LIN {X 60.580,Y -45.308,Z -141.426,A -90.000,B 90.000,C 0.000} C_DIS
LIN {X 60.651,Y -45.308,Z -141.391,A -90.000,B 90.000,C 0.000} C_DIS
LIN {X 60.882,Y -45.308,Z -141.285,A -90.000,B 90.000,C 0.000} C_DIS
LIN {X 61.927,Y -45.308,Z -140.871,A -90.000,B 90.000,C 0.000} C_DIS
LIN {X 63.864,Y -45.308,Z -140.277,A -90.000,B 90.000,C 0.000} C_DIS
LIN {X 64.038,Y -45.308,Z -140.235,A -90.000,B 90.000,C 0.000} C_DIS
LIN {X 65.559,Y -45.308,Z -140.294,A -90.000,B 90.000,C 0.000} C_DIS
LIN {X 65.640,Y -45.308,Z -140.321,A -90.000,B 90.000,C 0.000} C_DIS
LIN {X 66.939,Y -45.308,Z -140.767,A -90.000,B 90.000,C 0.000} C_DIS
LIN {X 67.087,Y -45.308,Z -140.867,A -90.000,B 90.000,C 0.000} C_DIS
LIN {X 67.673,Y -45.308,Z -141.467,A -90.000,B 90.000,C 0.000} C_DIS
LIN {X 67.788,Y -45.308,Z -141.605,A -90.000,B 90.000,C 0.000} C_DIS
LIN {X 68.275,Y -45.308,Z -142.438,A -90.000,B 90.000,C 0.000} C_DIS
LIN {X 68.917,Y -45.308,Z -143.399,A -90.000,B 90.000,C 0.000} C_DIS
LIN {X 68.990,Y -45.308,Z -143.563,A -90.000,B 90.000,C 0.000} C_DIS
LIN {X 69.573,Y -45.308,Z -144.914,A -90.000,B 90.000,C 0.000} C_DIS
LIN {X 69.855,Y -45.308,Z -145.939,A -90.000,B 90.000,C 0.000} C_DIS
LIN {X 69.892,Y -45.308,Z -146.103,A -90.000,B 90.000,C 0.000} C_DIS
LIN {X 69.904,Y -45.308,Z -146.218,A -90.000,B 90.000,C 0.000} C_DIS
LIN {X 70.372,Y -45.308,Z -149.844,A -90.000,B 90.000,C 0.000} C_DIS
LIN {X 70.397,Y -45.308,Z -150.079,A -90.000,B 90.000,C 0.000} C_DIS
LIN {X 70.477,Y -45.308,Z -152.363,A -90.000,B 90.000,C 0.000} C_DIS
LIN {X 70.544,Y -45.308,Z -153.906,A -90.000,B 90.000,C 0.000} C_DIS
LIN {X 70.353,Y -45.308,Z -157.725,A -90.000,B 90.000,C 0.000} C_DIS
LIN {X 70.338,Y -45.308,Z -157.908,A -90.000,B 90.000,C 0.000} C_DIS
LIN {X 70.199,Y -45.308,Z -158.814,A -90.000,B 90.000,C 0.000} C_DIS
LIN {X 69.684,Y -45.308,Z -161.585,A -90.000,B 90.000,C 0.000} C_DIS
LIN {X 69.620,Y -45.308,Z -161.813,A -90.000,B 90.000,C 0.000} C_DIS
LIN {X 69.546,Y -45.308,Z -162.065,A -90.000,B 90.000,C 0.000} C_DIS
LIN {X 68.616,Y -45.308,Z -165.294,A -90.000,B 90.000,C 0.000} C_DIS
LIN {X 68.534,Y -45.308,Z -165.522,A -90.000,B 90.000,C 0.000} C_DIS
LIN {X 67.458,Y -45.308,Z -168.597,A -90.000,B 90.000,C 0.000} C_DIS
LIN {X 66.943,Y -45.308,Z -170.008,A -90.000,B 90.000,C 0.000} C_DIS
LIN {X 66.324,Y -45.308,Z -171.617,A -90.000,B 90.000,C 0.000} C_DIS
LIN {X 66.282,Y -45.308,Z -171.733,A -90.000,B 90.000,C 0.000} C_DIS
LIN {X 65.339,Y -45.308,Z -174.575,A -90.000,B 90.000,C 0.000} C_DIS
LIN {X 64.922,Y -45.308,Z -176.632,A -90.000,B 90.000,C 0.000} C_DIS
LIN {X 64.757,Y -45.308,Z -177.363,A -90.000,B 90.000,C 0.000} C_DIS
LIN {X 64.366,Y -45.308,Z -180.088,A -90.000,B 90.000,C 0.000} C_DIS
LIN {X 64.330,Y -45.308,Z -180.550,A -90.000,B 90.000,C 0.000} C_DIS
LIN {X 64.152,Y -45.308,Z -182.594,A -90.000,B 90.000,C 0.000} C_DIS
LIN {X 64.105,Y -45.308,Z -183.519,A -90.000,B 90.000,C 0.000} C_DIS
LIN {X 63.918,Y -45.308,Z -186.609,A -90.000,B 90.000,C 0.000} C_DIS
LIN {X 63.839,Y -45.308,Z -187.772,A -90.000,B 90.000,C 0.000} C_DIS
LIN {X 63.829,Y -45.308,Z -187.892,A -90.000,B 90.000,C 0.000} C_DIS
LIN {X 63.562,Y -45.308,Z -190.517,A -90.000,B 90.000,C 0.000} C_DIS
LIN {X 63.102,Y -45.308,Z -193.390,A -90.000,B 90.000,C 0.000} C_DIS
LIN {X 62.752,Y -45.308,Z -194.947,A -90.000,B 90.000,C 0.000} C_DIS
LIN {X 62.328,Y -45.308,Z -196.733,A -90.000,B 90.000,C 0.000} C_DIS
LIN {X 62.297,Y -45.308,Z -196.846,A -90.000,B 90.000,C 0.000} C_DIS
LIN {X 61.644,Y -45.308,Z -199.064,A -90.000,B 90.000,C 0.000} C_DIS
LIN {X 61.144,Y -45.308,Z -200.631,A -90.000,B 90.000,C 0.000} C_DIS
LIN {X 59.629,Y -45.308,Z -204.936,A -90.000,B 90.000,C 0.000} C_DIS
LIN {X 59.533,Y -45.308,Z -205.201,A -90.000,B 90.000,C 0.000} C_DIS
LIN {X 57.775,Y -45.308,Z -209.890,A -90.000,B 90.000,C 0.000} C_DIS
LIN {X 55.827,Y -45.308,Z -214.869,A -90.000,B 90.000,C 0.000} C_DIS
LIN {X 54.437,Y -45.308,Z -218.314,A -90.000,B 90.000,C 0.000} C_DIS
LIN {X 53.740,Y -45.308,Z -220.037,A -90.000,B 90.000,C 0.000} C_DIS
LIN {X 52.345,Y -45.308,Z -223.157,A -90.000,B 90.000,C 0.000} C_DIS
LIN {X 51.395,Y -45.308,Z -225.293,A -90.000,B 90.000,C 0.000} C_DIS
LIN {X 49.882,Y -45.308,Z -228.183,A -90.000,B 90.000,C 0.000} C_DIS
LIN {X 48.676,Y -45.308,Z -230.534,A -90.000,B 90.000,C 0.000} C_DIS
LIN {X 48.535,Y -45.308,Z -230.778,A -90.000,B 90.000,C 0.000} C_DIS
LIN {X 46.664,Y -45.308,Z -233.707,A -90.000,B 90.000,C 0.000} C_DIS
LIN {X 45.317,Y -45.308,Z -235.896,A -90.000,B 90.000,C 0.000} C_DIS
LIN {X 42.480,Y -45.308,Z -239.403,A -90.000,B 90.000,C 0.000} C_DIS
LIN {X 41.445,Y -45.308,Z -240.753,A -90.000,B 90.000,C 0.000} C_DIS
LIN {X 41.263,Y -45.308,Z -240.969,A -90.000,B 90.000,C 0.000} C_DIS
LIN {X 38.792,Y -45.308,Z -243.561,A -90.000,B 90.000,C 0.000} C_DIS
LIN {X 38.792,Y -60.000,Z -243.561,A -90.000,B 90.000,C 0.000} C_DIS
LIN {X -67.298,Y -60.000,Z -243.561,A -90.000,B 90.000,C 0.000} C_DIS
LIN {X -67.298,Y -44.787,Z -243.561,A -90.000,B 90.000,C 0.000} C_DIS
LIN {X -67.270,Y -44.711,Z -243.409,A -90.000,B 90.000,C 0.000} C_DIS
LIN {X -67.144,Y -44.547,Z -243.047,A -90.000,B 90.000,C 0.000} C_DIS
LIN {X -67.046,Y -44.476,Z -242.863,A -90.000,B 90.000,C 0.000} C_DIS
LIN {X -66.669,Y -44.334,Z -242.397,A -90.000,B 90.000,C 0.000} C_DIS
LIN {X -66.161,Y -44.287,Z -242.036,A -90.000,B 90.000,C 0.000} C_DIS
LIN {X -65.652,Y -44.291,Z -241.768,A -90.000,B 90.000,C 0.000} C_DIS
LIN {X -64.439,Y -44.288,Z -241.140,A -90.000,B 90.000,C 0.000} C_DIS
LIN {X -60.910,Y -44.327,Z -239.407,A -90.000,B 90.000,C 0.000} C_DIS
LIN {X -57.171,Y -44.331,Z -237.595,A -90.000,B 90.000,C 0.000} C_DIS
LIN {X -55.898,Y -44.321,Z -236.982,A -90.000,B 90.000,C 0.000} C_DIS
LIN {X -55.409,Y -44.321,Z -236.755,A -90.000,B 90.000,C 0.000} C_DIS
LIN {X -54.668,Y -44.326,Z -236.421,A -90.000,B 90.000,C 0.000} C_DIS
LIN {X -52.760,Y -44.345,Z -235.573,A -90.000,B 90.000,C 0.000} C_DIS
LIN {X -49.209,Y -44.397,Z -234.093,A -90.000,B 90.000,C 0.000} C_DIS
LIN {X -47.684,Y -44.433,Z -233.484,A -90.000,B 90.000,C 0.000} C_DIS
LIN {X -45.954,Y -44.457,Z -232.802,A -90.000,B 90.000,C 0.000} C_DIS
LIN {X -45.316,Y -44.465,Z -232.551,A -90.000,B 90.000,C 0.000} C_DIS
LIN {X -44.202,Y -44.466,Z -232.120,A -90.000,B 90.000,C 0.000} C_DIS
LIN {X -41.863,Y -44.487,Z -231.267,A -90.000,B 90.000,C 0.000} C_DIS
LIN {X -41.293,Y -44.487,Z -231.062,A -90.000,B 90.000,C 0.000} C_DIS
LIN {X -39.930,Y -44.501,Z -230.603,A -90.000,B 90.000,C 0.000} C_DIS
LIN {X -39.608,Y -44.508,Z -230.503,A -90.000,B 90.000,C 0.000} C_DIS
LIN {X -38.618,Y -44.539,Z -230.217,A -90.000,B 90.000,C 0.000} C_DIS
LIN {X -37.408,Y -44.595,Z -229.897,A -90.000,B 90.000,C 0.000} C_DIS
LIN {X -36.049,Y -44.639,Z -229.528,A -90.000,B 90.000,C 0.000} C_DIS
LIN {X -34.932,Y -44.668,Z -229.228,A -90.000,B 90.000,C 0.000} C_DIS
LIN {X -34.798,Y -44.669,Z -229.193,A -90.000,B 90.000,C 0.000} C_DIS
LIN {X -34.317,Y -44.671,Z -229.068,A -90.000,B 90.000,C 0.000} C_DIS
LIN {X -32.516,Y -44.686,Z -228.647,A -90.000,B 90.000,C 0.000} C_DIS
LIN {X -32.064,Y -44.687,Z -228.542,A -90.000,B 90.000,C 0.000} C_DIS
LIN {X -31.983,Y -44.687,Z -228.525,A -90.000,B 90.000,C 0.000} C_DIS
LIN {X -30.904,Y -44.701,Z -228.321,A -90.000,B 90.000,C 0.000} C_DIS
LIN {X -30.738,Y -44.706,Z -228.296,A -90.000,B 90.000,C 0.000} C_DIS
LIN {X -29.560,Y -44.754,Z -228.178,A -90.000,B 90.000,C 0.000} C_DIS
LIN {X -29.093,Y -44.779,Z -228.147,A -90.000,B 90.000,C 0.000} C_DIS
LIN {X -28.473,Y -44.815,Z -228.106,A -90.000,B 90.000,C 0.000} C_DIS
LIN {X -27.647,Y -44.853,Z -228.056,A -90.000,B 90.000,C 0.000} C_DIS
LIN {X -27.097,Y -44.859,Z -228.027,A -90.000,B 90.000,C 0.000} C_DIS
LIN {X -26.119,Y -44.859,Z -227.944,A -90.000,B 90.000,C 0.000} C_DIS
LIN {X -25.569,Y -44.862,Z -227.908,A -90.000,B 90.000,C 0.000} C_DIS
LIN {X -25.234,Y -44.867,Z -227.901,A -90.000,B 90.000,C 0.000} C_DIS
LIN {X -25.053,Y -44.872,Z -227.906,A -90.000,B 90.000,C 0.000} C_DIS
LIN {X -24.470,Y -44.891,Z -227.950,A -90.000,B 90.000,C 0.000} C_DIS
LIN {X -24.240,Y -44.901,Z -227.981,A -90.000,B 90.000,C 0.000} C_DIS
LIN {X -23.242,Y -44.958,Z -228.173,A -90.000,B 90.000,C 0.000} C_DIS
LIN {X -23.055,Y -44.967,Z -228.209,A -90.000,B 90.000,C 0.000} C_DIS
LIN {X -22.552,Y -44.978,Z -228.310,A -90.000,B 90.000,C 0.000} C_DIS
LIN {X -22.026,Y -44.978,Z -228.417,A -90.000,B 90.000,C 0.000} C_DIS
LIN {X -21.725,Y -44.979,Z -228.487,A -90.000,B 90.000,C 0.000} C_DIS
LIN {X -20.617,Y -44.981,Z -228.753,A -90.000,B 90.000,C 0.000} C_DIS
LIN {X -20.425,Y -44.983,Z -228.813,A -90.000,B 90.000,C 0.000} C_DIS
LIN {X -20.250,Y -44.986,Z -228.873,A -90.000,B 90.000,C 0.000} C_DIS
LIN {X -20.100,Y -44.991,Z -228.938,A -90.000,B 90.000,C 0.000} C_DIS
LIN {X -20.052,Y -44.993,Z -228.962,A -90.000,B 90.000,C 0.000} C_DIS
LIN {X -19.857,Y -45.004,Z -229.077,A -90.000,B 90.000,C 0.000} C_DIS
LIN {X -19.708,Y -45.014,Z -229.176,A -90.000,B 90.000,C 0.000} C_DIS
LIN {X -19.467,Y -45.032,Z -229.343,A -90.000,B 90.000,C 0.000} C_DIS
LIN {X -19.339,Y -45.039,Z -229.432,A -90.000,B 90.000,C 0.000} C_DIS
LIN {X -18.431,Y -45.038,Z -230.074,A -90.000,B 90.000,C 0.000} C_DIS
LIN {X -17.329,Y -45.038,Z -230.904,A -90.000,B 90.000,C 0.000} C_DIS
LIN {X -17.131,Y -45.040,Z -231.074,A -90.000,B 90.000,C 0.000} C_DIS
LIN {X -16.995,Y -45.045,Z -231.222,A -90.000,B 90.000,C 0.000} C_DIS
LIN {X -16.869,Y -45.046,Z -231.372,A -90.000,B 90.000,C 0.000} C_DIS
LIN {X -16.752,Y -45.044,Z -231.533,A -90.000,B 90.000,C 0.000} C_DIS
LIN {X -15.804,Y -45.041,Z -233.094,A -90.000,B 90.000,C 0.000} C_DIS
LIN {X -15.426,Y -45.041,Z -233.734,A -90.000,B 90.000,C 0.000} C_DIS
LIN {X -15.257,Y -45.036,Z -234.022,A -90.000,B 90.000,C 0.000} C_DIS
LIN {X -15.172,Y -45.035,Z -234.182,A -90.000,B 90.000,C 0.000} C_DIS
LIN {X -14.961,Y -45.035,Z -234.654,A -90.000,B 90.000,C 0.000} C_DIS
LIN {X -14.274,Y -45.040,Z -236.188,A -90.000,B 90.000,C 0.000} C_DIS
LIN {X -14.110,Y -45.044,Z -236.552,A -90.000,B 90.000,C 0.000} C_DIS
LIN {X -13.993,Y -45.047,Z -236.794,A -90.000,B 90.000,C 0.000} C_DIS
LIN {X -13.255,Y -45.047,Z -238.011,A -90.000,B 90.000,C 0.000} C_DIS
LIN {X -13.065,Y -45.046,Z -238.296,A -90.000,B 90.000,C 0.000} C_DIS
LIN {X -12.733,Y -45.051,Z -238.794,A -90.000,B 90.000,C 0.000} C_DIS
LIN {X -12.646,Y -45.057,Z -238.923,A -90.000,B 90.000,C 0.000} C_DIS
LIN {X -11.097,Y -45.055,Z -240.071,A -90.000,B 90.000,C 0.000} C_DIS
LIN {X -10.769,Y -45.037,Z -240.129,A -90.000,B 90.000,C 0.000} C_DIS
LIN {X -10.257,Y -45.024,Z -240.217,A -90.000,B 90.000,C 0.000} C_DIS
LIN {X -9.508,Y -45.062,Z -240.340,A -90.000,B 90.000,C 0.000} C_DIS
LIN {X -8.784,Y -45.078,Z -240.341,A -90.000,B 90.000,C 0.000} C_DIS
LIN {X -8.272,Y -45.078,Z -240.344,A -90.000,B 90.000,C 0.000} C_DIS
LIN {X -4.569,Y -44.924,Z -239.042,A -90.000,B 90.000,C 0.000} C_DIS
LIN {X -3.870,Y -44.924,Z -238.791,A -90.000,B 90.000,C 0.000} C_DIS
LIN {X -2.390,Y -44.970,Z -238.252,A -90.000,B 90.000,C 0.000} C_DIS
LIN {X -0.853,Y -44.908,Z -236.956,A -90.000,B 90.000,C 0.000} C_DIS
LIN {X -0.001,Y -44.910,Z -236.229,A -90.000,B 90.000,C 0.000} C_DIS
LIN {X 1.219,Y -44.920,Z -235.229,A -90.000,B 90.000,C 0.000} C_DIS
LIN {X 2.676,Y -44.867,Z -233.519,A -90.000,B 90.000,C 0.000} C_DIS
LIN {X 4.369,Y -44.865,Z -231.510,A -90.000,B 90.000,C 0.000} C_DIS
LIN {X 4.575,Y -44.856,Z -231.211,A -90.000,B 90.000,C 0.000} C_DIS
LIN {X 4.834,Y -44.847,Z -230.835,A -90.000,B 90.000,C 0.000} C_DIS
LIN {X 6.303,Y -44.802,Z -228.671,A -90.000,B 90.000,C 0.000} C_DIS
LIN {X 7.363,Y -44.796,Z -227.098,A -90.000,B 90.000,C 0.000} C_DIS
LIN {X 7.515,Y -44.796,Z -226.878,A -90.000,B 90.000,C 0.000} C_DIS
LIN {X 7.864,Y -44.798,Z -226.373,A -90.000,B 90.000,C 0.000} C_DIS
LIN {X 7.939,Y -44.798,Z -226.259,A -90.000,B 90.000,C 0.000} C_DIS
LIN {X 9.938,Y -44.768,Z -222.971,A -90.000,B 90.000,C 0.000} C_DIS
LIN {X 10.445,Y -44.768,Z -222.134,A -90.000,B 90.000,C 0.000} C_DIS
LIN {X 10.596,Y -44.770,Z -221.883,A -90.000,B 90.000,C 0.000} C_DIS
LIN {X 11.790,Y -44.762,Z -219.763,A -90.000,B 90.000,C 0.000} C_DIS
LIN {X 12.145,Y -44.764,Z -219.132,A -90.000,B 90.000,C 0.000} C_DIS
LIN {X 12.682,Y -44.770,Z -218.203,A -90.000,B 90.000,C 0.000} C_DIS
LIN {X 13.008,Y -44.771,Z -217.642,A -90.000,B 90.000,C 0.000} C_DIS
LIN {X 13.171,Y -44.776,Z -217.358,A -90.000,B 90.000,C 0.000} C_DIS
LIN {X 14.056,Y -44.792,Z -215.663,A -90.000,B 90.000,C 0.000} C_DIS
LIN {X 14.543,Y -44.796,Z -214.696,A -90.000,B 90.000,C 0.000} C_DIS
LIN {X 15.364,Y -44.800,Z -213.069,A -90.000,B 90.000,C 0.000} C_DIS
LIN {X 15.477,Y -44.804,Z -212.843,A -90.000,B 90.000,C 0.000} C_DIS
LIN {X 15.756,Y -44.812,Z -212.254,A -90.000,B 90.000,C 0.000} C_DIS
LIN {X 16.265,Y -44.814,Z -211.045,A -90.000,B 90.000,C 0.000} C_DIS
LIN {X 17.100,Y -44.822,Z -209.043,A -90.000,B 90.000,C 0.000} C_DIS
LIN {X 17.373,Y -44.824,Z -208.357,A -90.000,B 90.000,C 0.000} C_DIS
LIN {X 18.130,Y -44.858,Z -206.146,A -90.000,B 90.000,C 0.000} C_DIS
LIN {X 18.726,Y -44.870,Z -204.142,A -90.000,B 90.000,C 0.000} C_DIS
LIN {X 18.849,Y -44.875,Z -203.668,A -90.000,B 90.000,C 0.000} C_DIS
LIN {X 18.987,Y -44.872,Z -202.926,A -90.000,B 90.000,C 0.000} C_DIS
LIN {X 19.274,Y -44.870,Z -201.502,A -90.000,B 90.000,C 0.000} C_DIS
LIN {X 19.608,Y -44.855,Z -199.853,A -90.000,B 90.000,C 0.000} C_DIS
LIN {X 19.652,Y -44.853,Z -199.630,A -90.000,B 90.000,C 0.000} C_DIS
LIN {X 20.199,Y -44.801,Z -196.858,A -90.000,B 90.000,C 0.000} C_DIS
LIN {X 20.446,Y -44.795,Z -195.895,A -90.000,B 90.000,C 0.000} C_DIS
LIN {X 20.541,Y -44.786,Z -195.535,A -90.000,B 90.000,C 0.000} C_DIS
LIN {X 20.564,Y -44.785,Z -195.453,A -90.000,B 90.000,C 0.000} C_DIS
LIN {X 20.642,Y -44.782,Z -195.202,A -90.000,B 90.000,C 0.000} C_DIS
LIN {X 20.915,Y -44.776,Z -194.417,A -90.000,B 90.000,C 0.000} C_DIS
LIN {X 21.045,Y -44.769,Z -194.046,A -90.000,B 90.000,C 0.000} C_DIS
LIN {X 21.881,Y -44.697,Z -191.473,A -90.000,B 90.000,C 0.000} C_DIS
LIN {X 21.929,Y -44.695,Z -191.339,A -90.000,B 90.000,C 0.000} C_DIS
LIN {X 22.045,Y -44.695,Z -191.060,A -90.000,B 90.000,C 0.000} C_DIS
LIN {X 22.081,Y -44.692,Z -190.980,A -90.000,B 90.000,C 0.000} C_DIS
LIN {X 23.068,Y -44.639,Z -188.911,A -90.000,B 90.000,C 0.000} C_DIS
LIN {X 23.201,Y -44.628,Z -188.607,A -90.000,B 90.000,C 0.000} C_DIS
LIN {X 23.652,Y -44.602,Z -187.566,A -90.000,B 90.000,C 0.000} C_DIS
LIN {X 23.710,Y -44.598,Z -187.454,A -90.000,B 90.000,C 0.000} C_DIS
LIN {X 23.765,Y -44.596,Z -187.361,A -90.000,B 90.000,C 0.000} C_DIS
LIN {X 24.257,Y -44.583,Z -186.557,A -90.000,B 90.000,C 0.000} C_DIS
LIN {X 24.363,Y -44.580,Z -186.390,A -90.000,B 90.000,C 0.000} C_DIS
LIN {X 24.685,Y -44.577,Z -185.899,A -90.000,B 90.000,C 0.000} C_DIS
LIN {X 25.700,Y -44.551,Z -184.374,A -90.000,B 90.000,C 0.000} C_DIS
LIN {X 25.827,Y -44.545,Z -184.186,A -90.000,B 90.000,C 0.000} C_DIS
LIN {X 25.890,Y -44.543,Z -184.098,A -90.000,B 90.000,C 0.000} C_DIS
LIN {X 26.870,Y -44.535,Z -182.791,A -90.000,B 90.000,C 0.000} C_DIS
LIN {X 27.875,Y -44.525,Z -181.522,A -90.000,B 90.000,C 0.000} C_DIS
LIN {X 29.146,Y -44.523,Z -179.964,A -90.000,B 90.000,C 0.000} C_DIS
LIN {X 29.462,Y -44.519,Z -179.579,A -90.000,B 90.000,C 0.000} C_DIS
LIN {X 29.729,Y -44.519,Z -179.251,A -90.000,B 90.000,C 0.000} C_DIS
LIN {X 31.269,Y -44.533,Z -177.449,A -90.000,B 90.000,C 0.000} C_DIS
LIN {X 31.603,Y -44.552,Z -177.048,A -90.000,B 90.000,C 0.000} C_DIS
LIN {X 32.293,Y -44.548,Z -176.059,A -90.000,B 90.000,C 0.000} C_DIS
LIN {X 32.817,Y -44.549,Z -175.350,A -90.000,B 90.000,C 0.000} C_DIS
LIN {X 33.023,Y -44.559,Z -175.065,A -90.000,B 90.000,C 0.000} C_DIS
LIN {X 33.889,Y -44.552,Z -173.666,A -90.000,B 90.000,C 0.000} C_DIS
LIN {X 34.095,Y -44.551,Z -173.349,A -90.000,B 90.000,C 0.000} C_DIS
LIN {X 34.249,Y -44.557,Z -173.110,A -90.000,B 90.000,C 0.000} C_DIS
LIN {X 35.410,Y -44.546,Z -171.078,A -90.000,B 90.000,C 0.000} C_DIS
LIN {X 35.530,Y -44.547,Z -170.877,A -90.000,B 90.000,C 0.000} C_DIS
LIN {X 36.271,Y -44.534,Z -169.531,A -90.000,B 90.000,C 0.000} C_DIS
LIN {X 36.563,Y -44.534,Z -169.025,A -90.000,B 90.000,C 0.000} C_DIS
LIN {X 36.810,Y -44.537,Z -168.598,A -90.000,B 90.000,C 0.000} C_DIS
LIN {X 37.039,Y -44.535,Z -168.171,A -90.000,B 90.000,C 0.000} C_DIS
LIN {X 38.276,Y -44.538,Z -166.002,A -90.000,B 90.000,C 0.000} C_DIS
LIN {X 38.520,Y -44.543,Z -165.572,A -90.000,B 90.000,C 0.000} C_DIS
LIN {X 39.176,Y -44.542,Z -164.346,A -90.000,B 90.000,C 0.000} C_DIS
LIN {X 39.927,Y -44.546,Z -163.021,A -90.000,B 90.000,C 0.000} C_DIS
LIN {X 40.188,Y -44.551,Z -162.557,A -90.000,B 90.000,C 0.000} C_DIS
LIN {X 41.605,Y -44.556,Z -159.932,A -90.000,B 90.000,C 0.000} C_DIS
LIN {X 41.932,Y -44.555,Z -159.355,A -90.000,B 90.000,C 0.000} C_DIS
LIN {X 42.596,Y -44.549,Z -158.159,A -90.000,B 90.000,C 0.000} C_DIS
LIN {X 43.799,Y -44.562,Z -156.119,A -90.000,B 90.000,C 0.000} C_DIS
LIN {X 44.380,Y -44.572,Z -155.158,A -90.000,B 90.000,C 0.000} C_DIS
LIN {X 45.309,Y -44.590,Z -153.649,A -90.000,B 90.000,C 0.000} C_DIS
LIN {X 45.559,Y -44.590,Z -153.247,A -90.000,B 90.000,C 0.000} C_DIS
LIN {X 45.740,Y -44.590,Z -152.957,A -90.000,B 90.000,C 0.000} C_DIS
LIN {X 45.907,Y -44.592,Z -152.695,A -90.000,B 90.000,C 0.000} C_DIS
LIN {X 46.546,Y -44.608,Z -151.741,A -90.000,B 90.000,C 0.000} C_DIS
LIN {X 47.431,Y -44.625,Z -150.425,A -90.000,B 90.000,C 0.000} C_DIS
LIN {X 47.669,Y -44.620,Z -150.076,A -90.000,B 90.000,C 0.000} C_DIS
LIN {X 47.901,Y -44.615,Z -149.738,A -90.000,B 90.000,C 0.000} C_DIS
LIN {X 48.068,Y -44.610,Z -149.499,A -90.000,B 90.000,C 0.000} C_DIS
LIN {X 48.191,Y -44.611,Z -149.343,A -90.000,B 90.000,C 0.000} C_DIS
LIN {X 49.907,Y -44.673,Z -147.377,A -90.000,B 90.000,C 0.000} C_DIS
LIN {X 50.941,Y -44.677,Z -146.211,A -90.000,B 90.000,C 0.000} C_DIS
LIN {X 51.066,Y -44.678,Z -146.074,A -90.000,B 90.000,C 0.000} C_DIS
LIN {X 51.221,Y -44.681,Z -145.909,A -90.000,B 90.000,C 0.000} C_DIS
LIN {X 51.436,Y -44.689,Z -145.695,A -90.000,B 90.000,C 0.000} C_DIS
LIN {X 51.619,Y -44.693,Z -145.513,A -90.000,B 90.000,C 0.000} C_DIS
LIN {X 52.346,Y -44.693,Z -144.801,A -90.000,B 90.000,C 0.000} C_DIS
LIN {X 52.988,Y -44.702,Z -144.207,A -90.000,B 90.000,C 0.000} C_DIS
LIN {X 53.091,Y -44.705,Z -144.118,A -90.000,B 90.000,C 0.000} C_DIS
LIN {X 53.267,Y -44.712,Z -143.975,A -90.000,B 90.000,C 0.000} C_DIS
LIN {X 54.172,Y -44.723,Z -143.252,A -90.000,B 90.000,C 0.000} C_DIS
LIN {X 54.518,Y -44.731,Z -142.974,A -90.000,B 90.000,C 0.000} C_DIS
LIN {X 54.749,Y -44.738,Z -142.797,A -90.000,B 90.000,C 0.000} C_DIS
LIN {X 54.837,Y -44.742,Z -142.733,A -90.000,B 90.000,C 0.000} C_DIS
LIN {X 55.082,Y -44.748,Z -142.568,A -90.000,B 90.000,C 0.000} C_DIS
LIN {X 55.785,Y -44.751,Z -142.100,A -90.000,B 90.000,C 0.000} C_DIS
LIN {X 56.241,Y -44.739,Z -141.749,A -90.000,B 90.000,C 0.000} C_DIS
LIN {X 56.322,Y -44.739,Z -141.685,A -90.000,B 90.000,C 0.000} C_DIS
LIN {X 56.542,Y -44.741,Z -141.520,A -90.000,B 90.000,C 0.000} C_DIS
LIN {X 56.749,Y -44.746,Z -141.382,A -90.000,B 90.000,C 0.000} C_DIS
LIN {X 57.457,Y -44.779,Z -140.972,A -90.000,B 90.000,C 0.000} C_DIS
LIN {X 58.083,Y -44.806,Z -140.612,A -90.000,B 90.000,C 0.000} C_DIS
LIN {X 58.544,Y -44.821,Z -140.347,A -90.000,B 90.000,C 0.000} C_DIS
LIN {X 59.599,Y -44.842,Z -139.747,A -90.000,B 90.000,C 0.000} C_DIS
LIN {X 59.775,Y -44.847,Z -139.653,A -90.000,B 90.000,C 0.000} C_DIS
LIN {X 60.047,Y -44.858,Z -139.523,A -90.000,B 90.000,C 0.000} C_DIS
LIN {X 60.145,Y -44.863,Z -139.480,A -90.000,B 90.000,C 0.000} C_DIS
LIN {X 61.205,Y -44.906,Z -139.050,A -90.000,B 90.000,C 0.000} C_DIS
LIN {X 61.325,Y -44.912,Z -139.006,A -90.000,B 90.000,C 0.000} C_DIS
LIN {X 63.019,Y -44.951,Z -138.478,A -90.000,B 90.000,C 0.000} C_DIS
LIN {X 63.286,Y -44.961,Z -138.394,A -90.000,B 90.000,C 0.000} C_DIS
LIN {X 63.399,Y -44.965,Z -138.362,A -90.000,B 90.000,C 0.000} C_DIS
LIN {X 63.573,Y -44.973,Z -138.319,A -90.000,B 90.000,C 0.000} C_DIS
LIN {X 63.859,Y -44.990,Z -138.268,A -90.000,B 90.000,C 0.000} C_DIS
LIN {X 63.954,Y -44.996,Z -138.261,A -90.000,B 90.000,C 0.000} C_DIS
LIN {X 64.116,Y -45.010,Z -138.259,A -90.000,B 90.000,C 0.000} C_DIS
LIN {X 64.331,Y -45.029,Z -138.264,A -90.000,B 90.000,C 0.000} C_DIS
LIN {X 64.863,Y -45.047,Z -138.283,A -90.000,B 90.000,C 0.000} C_DIS
LIN {X 65.684,Y -45.048,Z -138.315,A -90.000,B 90.000,C 0.000} C_DIS
LIN {X 66.179,Y -45.057,Z -138.410,A -90.000,B 90.000,C 0.000} C_DIS
LIN {X 67.117,Y -45.087,Z -138.726,A -90.000,B 90.000,C 0.000} C_DIS
LIN {X 67.287,Y -45.088,Z -138.785,A -90.000,B 90.000,C 0.000} C_DIS
LIN {X 67.593,Y -45.077,Z -138.891,A -90.000,B 90.000,C 0.000} C_DIS
LIN {X 67.764,Y -45.067,Z -138.961,A -90.000,B 90.000,C 0.000} C_DIS
LIN {X 68.013,Y -45.053,Z -139.099,A -90.000,B 90.000,C 0.000} C_DIS
LIN {X 68.201,Y -45.047,Z -139.227,A -90.000,B 90.000,C 0.000} C_DIS
LIN {X 68.448,Y -45.041,Z -139.426,A -90.000,B 90.000,C 0.000} C_DIS
LIN {X 68.506,Y -45.041,Z -139.483,A -90.000,B 90.000,C 0.000} C_DIS
LIN {X 69.091,Y -45.041,Z -140.082,A -90.000,B 90.000,C 0.000} C_DIS
LIN {X 69.156,Y -45.042,Z -140.153,A -90.000,B 90.000,C 0.000} C_DIS
LIN {X 69.272,Y -45.041,Z -140.290,A -90.000,B 90.000,C 0.000} C_DIS
LIN {X 69.341,Y -45.039,Z -140.373,A -90.000,B 90.000,C 0.000} C_DIS
LIN {X 69.430,Y -45.037,Z -140.496,A -90.000,B 90.000,C 0.000} C_DIS
LIN {X 69.500,Y -45.036,Z -140.608,A -90.000,B 90.000,C 0.000} C_DIS
LIN {X 69.955,Y -45.036,Z -141.387,A -90.000,B 90.000,C 0.000} C_DIS
LIN {X 70.098,Y -45.033,Z -141.602,A -90.000,B 90.000,C 0.000} C_DIS
LIN {X 70.558,Y -44.991,Z -142.301,A -90.000,B 90.000,C 0.000} C_DIS
LIN {X 70.720,Y -44.976,Z -142.599,A -90.000,B 90.000,C 0.000} C_DIS
LIN {X 70.739,Y -44.975,Z -142.643,A -90.000,B 90.000,C 0.000} C_DIS
LIN {X 71.371,Y -44.909,Z -144.137,A -90.000,B 90.000,C 0.000} C_DIS
LIN {X 71.460,Y -44.902,Z -144.393,A -90.000,B 90.000,C 0.000} C_DIS
LIN {X 71.742,Y -44.891,Z -145.423,A -90.000,B 90.000,C 0.000} C_DIS
LIN {X 71.765,Y -44.890,Z -145.517,A -90.000,B 90.000,C 0.000} C_DIS
LIN {X 71.801,Y -44.890,Z -145.681,A -90.000,B 90.000,C 0.000} C_DIS
LIN {X 71.836,Y -44.893,Z -145.886,A -90.000,B 90.000,C 0.000} C_DIS
LIN {X 71.845,Y -44.894,Z -145.968,A -90.000,B 90.000,C 0.000} C_DIS
LIN {X 71.894,Y -44.901,Z -146.336,A -90.000,B 90.000,C 0.000} C_DIS
LIN {X 72.312,Y -44.890,Z -149.594,A -90.000,B 90.000,C 0.000} C_DIS
LIN {X 72.342,Y -44.890,Z -149.873,A -90.000,B 90.000,C 0.000} C_DIS
LIN {X 72.352,Y -44.891,Z -150.010,A -90.000,B 90.000,C 0.000} C_DIS
LIN {X 72.365,Y -44.896,Z -150.357,A -90.000,B 90.000,C 0.000} C_DIS
LIN {X 72.425,Y -44.862,Z -152.273,A -90.000,B 90.000,C 0.000} C_DIS
LIN {X 72.484,Y -44.830,Z -153.823,A -90.000,B 90.000,C 0.000} C_DIS
LIN {X 72.483,Y -44.829,Z -154.003,A -90.000,B 90.000,C 0.000} C_DIS
LIN {X 72.473,Y -44.829,Z -154.206,A -90.000,B 90.000,C 0.000} C_DIS
LIN {X 72.280,Y -44.780,Z -157.815,A -90.000,B 90.000,C 0.000} C_DIS
LIN {X 72.259,Y -44.778,Z -158.070,A -90.000,B 90.000,C 0.000} C_DIS
LIN {X 72.244,Y -44.778,Z -158.201,A -90.000,B 90.000,C 0.000} C_DIS
LIN {X 72.103,Y -44.771,Z -159.107,A -90.000,B 90.000,C 0.000} C_DIS
LIN {X 71.586,Y -44.771,Z -161.895,A -90.000,B 90.000,C 0.000} C_DIS
LIN {X 71.567,Y -44.769,Z -161.987,A -90.000,B 90.000,C 0.000} C_DIS
LIN {X 71.533,Y -44.768,Z -162.121,A -90.000,B 90.000,C 0.000} C_DIS
LIN {X 71.395,Y -44.767,Z -162.602,A -90.000,B 90.000,C 0.000} C_DIS
LIN {X 70.529,Y -44.765,Z -165.605,A -90.000,B 90.000,C 0.000} C_DIS
LIN {X 70.465,Y -44.761,Z -165.826,A -90.000,B 90.000,C 0.000} C_DIS
LIN {X 70.427,Y -44.760,Z -165.943,A -90.000,B 90.000,C 0.000} C_DIS
LIN {X 70.347,Y -44.760,Z -166.164,A -90.000,B 90.000,C 0.000} C_DIS
LIN {X 69.884,Y -44.757,Z -167.486,A -90.000,B 90.000,C 0.000} C_DIS
LIN {X 69.386,Y -44.757,Z -168.908,A -90.000,B 90.000,C 0.000} C_DIS
LIN {X 69.272,Y -44.755,Z -169.232,A -90.000,B 90.000,C 0.000} C_DIS
LIN {X 68.748,Y -44.753,Z -170.667,A -90.000,B 90.000,C 0.000} C_DIS
LIN {X 68.220,Y -44.759,Z -172.045,A -90.000,B 90.000,C 0.000} C_DIS
LIN {X 68.100,Y -44.764,Z -172.364,A -90.000,B 90.000,C 0.000} C_DIS
LIN {X 67.259,Y -44.767,Z -174.903,A -90.000,B 90.000,C 0.000} C_DIS
LIN {X 67.204,Y -44.771,Z -175.071,A -90.000,B 90.000,C 0.000} C_DIS
LIN {X 66.811,Y -44.762,Z -176.996,A -90.000,B 90.000,C 0.000} C_DIS
LIN {X 66.651,Y -44.763,Z -177.711,A -90.000,B 90.000,C 0.000} C_DIS
LIN {X 66.420,Y -44.767,Z -179.327,A -90.000,B 90.000,C 0.000} C_DIS
LIN {X 66.281,Y -44.767,Z -180.299,A -90.000,B 90.000,C 0.000} C_DIS
LIN {X 66.272,Y -44.765,Z -180.412,A -90.000,B 90.000,C 0.000} C_DIS
LIN {X 66.077,Y -44.769,Z -182.692,A -90.000,B 90.000,C 0.000} C_DIS
LIN {X 66.063,Y -44.768,Z -182.930,A -90.000,B 90.000,C 0.000} C_DIS
LIN {X 66.029,Y -44.768,Z -183.603,A -90.000,B 90.000,C 0.000} C_DIS
LIN {X 65.918,Y -44.772,Z -185.458,A -90.000,B 90.000,C 0.000} C_DIS
LIN {X 65.848,Y -44.769,Z -186.602,A -90.000,B 90.000,C 0.000} C_DIS
LIN {X 65.772,Y -44.765,Z -187.735,A -90.000,B 90.000,C 0.000} C_DIS
LIN {X 65.745,Y -44.760,Z -188.054,A -90.000,B 90.000,C 0.000} C_DIS
LIN {X 65.460,Y -44.708,Z -190.715,A -90.000,B 90.000,C 0.000} C_DIS
LIN {X 65.446,Y -44.706,Z -190.818,A -90.000,B 90.000,C 0.000} C_DIS
LIN {X 65.426,Y -44.706,Z -190.942,A -90.000,B 90.000,C 0.000} C_DIS
LIN {X 65.314,Y -44.693,Z -191.614,A -90.000,B 90.000,C 0.000} C_DIS
LIN {X 64.970,Y -44.658,Z -193.689,A -90.000,B 90.000,C 0.000} C_DIS
LIN {X 64.947,Y -44.657,Z -193.806,A -90.000,B 90.000,C 0.000} C_DIS
LIN {X 64.588,Y -44.634,Z -195.361,A -90.000,B 90.000,C 0.000} C_DIS
LIN {X 64.158,Y -44.617,Z -197.149,A -90.000,B 90.000,C 0.000} C_DIS
LIN {X 64.118,Y -44.614,Z -197.297,A -90.000,B 90.000,C 0.000} C_DIS
LIN {X 63.435,Y -44.594,Z -199.592,A -90.000,B 90.000,C 0.000} C_DIS
LIN {X 63.229,Y -44.594,Z -200.242,A -90.000,B 90.000,C 0.000} C_DIS
LIN {X 62.984,Y -44.594,Z -201.009,A -90.000,B 90.000,C 0.000} C_DIS
LIN {X 62.923,Y -44.592,Z -201.198,A -90.000,B 90.000,C 0.000} C_DIS
LIN {X 61.464,Y -44.590,Z -205.345,A -90.000,B 90.000,C 0.000} C_DIS
LIN {X 61.299,Y -44.589,Z -205.805,A -90.000,B 90.000,C 0.000} C_DIS
LIN {X 59.522,Y -44.587,Z -210.545,A -90.000,B 90.000,C 0.000} C_DIS
LIN {X 57.563,Y -44.586,Z -215.548,A -90.000,B 90.000,C 0.000} C_DIS
LIN {X 56.526,Y -44.585,Z -218.119,A -90.000,B 90.000,C 0.000} C_DIS
LIN {X 55.553,Y -44.585,Z -220.526,A -90.000,B 90.000,C 0.000} C_DIS
LIN {X 55.467,Y -44.582,Z -220.736,A -90.000,B 90.000,C 0.000} C_DIS
LIN {X 54.511,Y -44.582,Z -222.879,A -90.000,B 90.000,C 0.000} C_DIS
LIN {X 53.209,Y -44.583,Z -225.799,A -90.000,B 90.000,C 0.000} C_DIS
LIN {X 53.095,Y -44.577,Z -226.050,A -90.000,B 90.000,C 0.000} C_DIS
LIN {X 53.057,Y -44.576,Z -226.130,A -90.000,B 90.000,C 0.000} C_DIS
LIN {X 51.538,Y -44.585,Z -229.041,A -90.000,B 90.000,C 0.000} C_DIS
LIN {X 50.499,Y -44.585,Z -231.064,A -90.000,B 90.000,C 0.000} C_DIS
LIN {X 50.431,Y -44.582,Z -231.194,A -90.000,B 90.000,C 0.000} C_DIS
LIN {X 50.303,Y -44.576,Z -231.436,A -90.000,B 90.000,C 0.000} C_DIS
LIN {X 50.122,Y -44.572,Z -231.747,A -90.000,B 90.000,C 0.000} C_DIS
LIN {X 48.254,Y -44.592,Z -234.687,A -90.000,B 90.000,C 0.000} C_DIS
LIN {X 47.161,Y -44.592,Z -236.462,A -90.000,B 90.000,C 0.000} C_DIS
LIN {X 46.922,Y -44.572,Z -236.836,A -90.000,B 90.000,C 0.000} C_DIS
LIN {X 46.845,Y -44.568,Z -236.954,A -90.000,B 90.000,C 0.000} C_DIS
LIN {X 46.776,Y -44.568,Z -237.046,A -90.000,B 90.000,C 0.000} C_DIS
LIN {X 43.977,Y -44.606,Z -240.530,A -90.000,B 90.000,C 0.000} C_DIS
LIN {X 43.325,Y -44.606,Z -241.379,A -90.000,B 90.000,C 0.000} C_DIS
LIN {X 43.161,Y -44.602,Z -241.591,A -90.000,B 90.000,C 0.000} C_DIS
LIN {X 42.926,Y -44.589,Z -241.888,A -90.000,B 90.000,C 0.000} C_DIS
LIN {X 42.871,Y -44.586,Z -241.956,A -90.000,B 90.000,C 0.000} C_DIS
LIN {X 42.687,Y -44.580,Z -242.170,A -90.000,B 90.000,C 0.000} C_DIS
LIN {X 42.611,Y -44.579,Z -242.254,A -90.000,B 90.000,C 0.000} C_DIS
LIN {X 41.925,Y -44.579,Z -242.974,A -90.000,B 90.000,C 0.000} C_DIS
LIN {X 41.369,Y -44.587,Z -243.561,A -90.000,B 90.000,C 0.000} C_DIS
LIN {X 41.369,Y -60.000,Z -243.561,A -90.000,B 90.000,C 0.000} C_DIS
LIN {X -56.008,Y -60.000,Z -235.133,A -90.000,B 90.000,C 0.000} C_DIS
LIN {X -56.008,Y -43.308,Z -235.133,A -90.000,B 90.000,C 0.000} C_DIS
LIN {X -55.361,Y -43.318,Z -234.839,A -90.000,B 90.000,C 0.000} C_DIS
LIN {X -53.415,Y -43.352,Z -233.966,A -90.000,B 90.000,C 0.000} C_DIS
LIN {X -52.543,Y -43.378,Z -233.594,A -90.000,B 90.000,C 0.000} C_DIS
LIN {X -51.053,Y -43.410,Z -232.966,A -90.000,B 90.000,C 0.000} C_DIS
LIN {X -49.827,Y -43.429,Z -232.455,A -90.000,B 90.000,C 0.000} C_DIS
LIN {X -45.890,Y -43.522,Z -230.883,A -90.000,B 90.000,C 0.000} C_DIS
LIN {X -44.802,Y -43.537,Z -230.453,A -90.000,B 90.000,C 0.000} C_DIS
LIN {X -41.858,Y -43.612,Z -229.355,A -90.000,B 90.000,C 0.000} C_DIS
LIN {X -40.787,Y -43.652,Z -228.979,A -90.000,B 90.000,C 0.000} C_DIS
LIN {X -40.453,Y -43.666,Z -228.862,A -90.000,B 90.000,C 0.000} C_DIS
LIN {X -40.090,Y -43.683,Z -228.746,A -90.000,B 90.000,C 0.000} C_DIS
LIN {X -39.516,Y -43.713,Z -228.574,A -90.000,B 90.000,C 0.000} C_DIS
LIN {X -39.050,Y -43.730,Z -228.439,A -90.000,B 90.000,C 0.000} C_DIS
LIN {X -37.852,Y -43.785,Z -228.123,A -90.000,B 90.000,C 0.000} C_DIS
LIN {X -35.704,Y -43.873,Z -227.532,A -90.000,B 90.000,C 0.000} C_DIS
LIN {X -34.731,Y -43.905,Z -227.267,A -90.000,B 90.000,C 0.000} C_DIS
LIN {X -32.446,Y -44.000,Z -226.703,A -90.000,B 90.000,C 0.000} C_DIS
LIN {X -32.324,Y -44.006,Z -226.676,A -90.000,B 90.000,C 0.000} C_DIS
LIN {X -31.694,Y -44.042,Z -226.547,A -90.000,B 90.000,C 0.000} C_DIS
LIN {X -31.250,Y -44.067,Z -226.456,A -90.000,B 90.000,C 0.000} C_DIS
LIN {X -31.001,Y -44.085,Z -226.413,A -90.000,B 90.000,C 0.000} C_DIS
LIN {X -30.903,Y -44.093,Z -226.399,A -90.000,B 90.000,C 0.000} C_DIS
LIN {X -30.749,Y -44.102,Z -226.383,A -90.000,B 90.000,C 0.000} C_DIS
LIN {X -29.657,Y -44.157,Z -226.272,A -90.000,B 90.000,C 0.000} C_DIS
LIN {X -28.562,Y -44.223,Z -226.198,A -90.000,B 90.000,C 0.000} C_DIS
LIN {X -27.339,Y -44.297,Z -226.117,A -90.000,B 90.000,C 0.000} C_DIS
LIN {X -27.223,Y -44.303,Z -226.110,A -90.000,B 90.000,C 0.000} C_DIS
LIN {X -26.196,Y -44.349,Z -226.011,A -90.000,B 90.000,C 0.000} C_DIS
LIN {X -25.626,Y -44.379,Z -225.968,A -90.000,B 90.000,C 0.000} C_DIS
LIN {X -25.219,Y -44.401,Z -225.956,A -90.000,B 90.000,C 0.000} C_DIS
LIN {X -24.916,Y -44.422,Z -225.962,A -90.000,B 90.000,C 0.000} C_DIS
LIN {X -24.803,Y -44.431,Z -225.970,A -90.000,B 90.000,C 0.000} C_DIS
LIN {X -24.278,Y -44.451,Z -226.009,A -90.000,B 90.000,C 0.000} C_DIS
LIN {X -23.941,Y -44.467,Z -226.051,A -90.000,B 90.000,C 0.000} C_DIS
LIN {X -23.762,Y -44.478,Z -226.083,A -90.000,B 90.000,C 0.000} C_DIS
LIN {X -21.576,Y -44.604,Z -226.504,A -90.000,B 90.000,C 0.000} C_DIS
LIN {X -21.265,Y -44.624,Z -226.574,A -90.000,B 90.000,C 0.000} C_DIS
LIN {X -20.982,Y -44.639,Z -226.639,A -90.000,B 90.000,C 0.000} C_DIS
LIN {X -20.471,Y -44.653,Z -226.759,A -90.000,B 90.000,C 0.000} C_DIS
LIN {X -20.157,Y -44.655,Z -226.834,A -90.000,B 90.000,C 0.000} C_DIS
LIN {X -20.020,Y -44.658,Z -226.871,A -90.000,B 90.000,C 0.000} C_DIS
LIN {X -19.768,Y -44.663,Z -226.951,A -90.000,B 90.000,C 0.000} C_DIS
LIN {X -19.594,Y -44.667,Z -227.011,A -90.000,B 90.000,C 0.000} C_DIS
LIN {X -19.497,Y -44.670,Z -227.047,A -90.000,B 90.000,C 0.000} C_DIS
LIN {X -19.281,Y -44.678,Z -227.140,A -90.000,B 90.000,C 0.000} C_DIS
LIN {X -19.160,Y -44.684,Z -227.199,A -90.000,B 90.000,C 0.000} C_DIS
LIN {X -19.089,Y -44.687,Z -227.236,A -90.000,B 90.000,C 0.000} C_DIS
LIN {X -18.836,Y -44.702,Z -227.384,A -90.000,B 90.000,C 0.000} C_DIS
LIN {X -18.671,Y -44.714,Z -227.490,A -90.000,B 90.000,C 0.000} C_DIS
LIN {X -18.447,Y -44.730,Z -227.643,A -90.000,B 90.000,C 0.000} C_DIS
LIN {X -17.850,Y -44.775,Z -228.057,A -90.000,B 90.000,C 0.000} C_DIS
LIN {X -17.721,Y -44.781,Z -228.147,A -90.000,B 90.000,C 0.000} C_DIS
LIN {X -17.238,Y -44.781,Z -228.489,A -90.000,B 90.000,C 0.000} C_DIS
LIN {X -16.136,Y -44.782,Z -229.319,A -90.000,B 90.000,C 0.000} C_DIS
LIN {X -16.033,Y -44.782,Z -229.402,A -90.000,B 90.000,C 0.000} C_DIS
LIN {X -15.835,Y -44.784,Z -229.572,A -90.000,B 90.000,C 0.000} C_DIS
LIN {X -15.690,Y -44.787,Z -229.711,A -90.000,B 90.000,C 0.000} C_DIS
LIN {X -15.533,Y -44.792,Z -229.881,A -90.000,B 90.000,C 0.000} C_DIS
LIN {X -15.451,Y -44.796,Z -229.975,A -90.000,B 90.000,C 0.000} C_DIS
LIN {X -15.336,Y -44.796,Z -230.112,A -90.000,B 90.000,C 0.000} C_DIS
LIN {X -15.269,Y -44.793,Z -230.200,A -90.000,B 90.000,C 0.000} C_DIS
LIN {X -15.152,Y -44.789,Z -230.360,A -90.000,B 90.000,C 0.000} C_DIS
LIN {X -15.056,Y -44.787,Z -230.504,A -90.000,B 90.000,C 0.000} C_DIS
LIN {X -14.501,Y -44.776,Z -231.422,A -90.000,B 90.000,C 0.000} C_DIS
LIN {X -14.098,Y -44.775,Z -232.086,A -90.000,B 90.000,C 0.000} C_DIS
LIN {X -13.890,Y -44.774,Z -232.438,A -90.000,B 90.000,C 0.000} C_DIS
LIN {X -13.598,Y -44.767,Z -232.934,A -90.000,B 90.000,C 0.000} C_DIS
LIN {X -13.547,Y -44.766,Z -233.021,A -90.000,B 90.000,C 0.000} C_DIS
LIN {X -13.414,Y -44.765,Z -233.268,A -90.000,B 90.000,C 0.000} C_DIS
LIN {X -13.364,Y -44.765,Z -233.371,A -90.000,B 90.000,C 0.000} C_DIS
LIN {X -12.618,Y -44.773,Z -235.036,A -90.000,B 90.000,C 0.000} C_DIS
LIN {X -12.312,Y -44.785,Z -235.717,A -90.000,B 90.000,C 0.000} C_DIS
LIN {X -12.247,Y -44.787,Z -235.851,A -90.000,B 90.000,C 0.000} C_DIS
LIN {X -12.160,Y -44.787,Z -235.993,A -90.000,B 90.000,C 0.000} C_DIS
LIN {X -11.579,Y -44.802,Z -236.946,A -90.000,B 90.000,C 0.000} C_DIS
LIN {X -11.233,Y -44.808,Z -237.465,A -90.000,B 90.000,C 0.000} C_DIS
LIN {X -11.186,Y -44.811,Z -237.535,A -90.000,B 90.000,C 0.000} C_DIS
LIN {X -10.296,Y -44.811,Z -238.194,A -90.000,B 90.000,C 0.000} C_DIS
LIN {X -10.132,Y -44.801,Z -238.223,A -90.000,B 90.000,C 0.000} C_DIS
LIN {X -9.335,Y -44.782,Z -238.360,A -90.000,B 90.000,C 0.000} C_DIS
LIN {X -8.611,Y -44.753,Z -238.369,A -90.000,B 90.000,C 0.000} C_DIS
LIN {X -8.113,Y -44.713,Z -238.197,A -90.000,B 90.000,C 0.000} C_DIS
LIN {X -6.122,Y -44.631,Z -237.497,A -90.000,B 90.000,C 0.000} C_DIS
LIN {X -3.794,Y -44.610,Z -236.666,A -90.000,B 90.000,C 0.000} C_DIS
LIN {X -3.394,Y -44.623,Z -236.520,A -90.000,B 90.000,C 0.000} C_DIS
LIN {X -1.244,Y -44.538,Z -234.707,A -90.000,B 90.000,C 0.000} C_DIS
LIN {X -0.656,Y -44.519,Z -234.230,A -90.000,B 90.000,C 0.000} C_DIS
LIN {X -0.339,Y -44.513,Z -233.973,A -90.000,B 90.000,C 0.000} C_DIS
LIN {X -0.161,Y -44.516,Z -233.827,A -90.000,B 90.000,C 0.000} C_DIS
LIN {X 2.815,Y -44.409,Z -230.331,A -90.000,B 90.000,C 0.000} C_DIS
LIN {X 3.065,Y -44.392,Z -229.972,A -90.000,B 90.000,C 0.000} C_DIS
LIN {X 4.406,Y -44.354,Z -227.999,A -90.000,B 90.000,C 0.000} C_DIS
LIN {X 5.766,Y -44.315,Z -225.995,A -90.000,B 90.000,C 0.000} C_DIS
LIN {X 5.942,Y -44.312,Z -225.742,A -90.000,B 90.000,C 0.000} C_DIS
LIN {X 6.278,Y -44.311,Z -225.254,A -90.000,B 90.000,C 0.000} C_DIS
LIN {X 6.791,Y -44.297,Z -224.416,A -90.000,B 90.000,C 0.000} C_DIS
LIN {X 8.668,Y -44.280,Z -221.323,A -90.000,B 90.000,C 0.000} C_DIS
LIN {X 8.923,Y -44.285,Z -220.900,A -90.000,B 90.000,C 0.000} C_DIS
LIN {X 9.741,Y -44.288,Z -219.444,A -90.000,B 90.000,C 0.000} C_DIS
LIN {X 10.467,Y -44.279,Z -218.158,A -90.000,B 90.000,C 0.000} C_DIS
LIN {X 11.210,Y -44.276,Z -216.879,A -90.000,B 90.000,C 0.000} C_DIS
LIN {X 11.473,Y -44.286,Z -216.421,A -90.000,B 90.000,C 0.000} C_DIS
LIN {X 12.353,Y -44.297,Z -214.737,A -90.000,B 90.000,C 0.000} C_DIS
LIN {X 12.438,Y -44.297,Z -214.567,A -90.000,B 90.000,C 0.000} C_DIS
LIN {X 13.521,Y -44.334,Z -212.403,A -90.000,B 90.000,C 0.000} C_DIS
LIN {X 13.729,Y -44.345,Z -211.985,A -90.000,B 90.000,C 0.000} C_DIS
LIN {X 13.979,Y -44.357,Z -211.456,A -90.000,B 90.000,C 0.000} C_DIS
LIN {X 14.466,Y -44.373,Z -210.290,A -90.000,B 90.000,C 0.000} C_DIS
LIN {X 15.289,Y -44.404,Z -208.303,A -90.000,B 90.000,C 0.000} C_DIS
LIN {X 15.461,Y -44.410,Z -207.870,A -90.000,B 90.000,C 0.000} C_DIS
LIN {X 15.539,Y -44.415,Z -207.672,A -90.000,B 90.000,C 0.000} C_DIS
LIN {X 16.267,Y -44.443,Z -205.546,A -90.000,B 90.000,C 0.000} C_DIS
LIN {X 16.843,Y -44.451,Z -203.614,A -90.000,B 90.000,C 0.000} C_DIS
LIN {X 16.940,Y -44.451,Z -203.242,A -90.000,B 90.000,C 0.000} C_DIS
LIN {X 17.073,Y -44.441,Z -202.541,A -90.000,B 90.000,C 0.000} C_DIS
LIN {X 17.564,Y -44.413,Z -200.127,A -90.000,B 90.000,C 0.000} C_DIS
LIN {X 17.720,Y -44.392,Z -199.373,A -90.000,B 90.000,C 0.000} C_DIS
LIN {X 17.850,Y -44.371,Z -198.723,A -90.000,B 90.000,C 0.000} C_DIS
LIN {X 18.306,Y -44.272,Z -196.484,A -90.000,B 90.000,C 0.000} C_DIS
LIN {X 18.331,Y -44.268,Z -196.381,A -90.000,B 90.000,C 0.000} C_DIS
LIN {X 18.693,Y -44.226,Z -195.015,A -90.000,B 90.000,C 0.000} C_DIS
LIN {X 18.732,Y -44.223,Z -194.882,A -90.000,B 90.000,C 0.000} C_DIS
LIN {X 18.830,Y -44.212,Z -194.575,A -90.000,B 90.000,C 0.000} C_DIS
LIN {X 19.230,Y -44.181,Z -193.446,A -90.000,B 90.000,C 0.000} C_DIS
LIN {X 19.272,Y -44.176,Z -193.320,A -90.000,B 90.000,C 0.000} C_DIS
LIN {X 20.103,Y -44.035,Z -190.839,A -90.000,B 90.000,C 0.000} C_DIS
LIN {X 20.155,Y -44.029,Z -190.700,A -90.000,B 90.000,C 0.000} C_DIS
LIN {X 20.189,Y -44.026,Z -190.616,A -90.000,B 90.000,C 0.000} C_DIS
LIN {X 20.340,Y -44.017,Z -190.265,A -90.000,B 90.000,C 0.000} C_DIS
LIN {X 20.376,Y -44.014,Z -190.185,A -90.000,B 90.000,C 0.000} C_DIS
LIN {X 21.365,Y -43.910,Z -188.156,A -90.000,B 90.000,C 0.000} C_DIS
LIN {X 21.667,Y -43.868,Z -187.485,A -90.000,B 90.000,C 0.000} C_DIS
LIN {X 21.912,Y -43.840,Z -186.933,A -90.000,B 90.000,C 0.000} C_DIS
LIN {X 21.961,Y -43.834,Z -186.823,A -90.000,B 90.000,C 0.000} C_DIS
LIN {X 22.069,Y -43.827,Z -186.610,A -90.000,B 90.000,C 0.000} C_DIS
LIN {X 22.173,Y -43.823,Z -186.429,A -90.000,B 90.000,C 0.000} C_DIS
LIN {X 22.775,Y -43.793,Z -185.462,A -90.000,B 90.000,C 0.000} C_DIS
LIN {X 23.162,Y -43.769,Z -184.884,A -90.000,B 90.000,C 0.000} C_DIS
LIN {X 24.098,Y -43.718,Z -183.502,A -90.000,B 90.000,C 0.000} C_DIS
LIN {X 24.342,Y -43.701,Z -183.147,A -90.000,B 90.000,C 0.000} C_DIS
LIN {X 24.448,Y -43.697,Z -183.001,A -90.000,B 90.000,C 0.000} C_DIS
LIN {X 24.690,Y -43.690,Z -182.682,A -90.000,B 90.000,C 0.000} C_DIS
LIN {X 25.459,Y -43.655,Z -181.680,A -90.000,B 90.000,C 0.000} C_DIS
LIN {X 26.489,Y -43.628,Z -180.392,A -90.000,B 90.000,C 0.000} C_DIS
LIN {X 27.452,Y -43.613,Z -179.223,A -90.000,B 90.000,C 0.000} C_DIS
LIN {X 27.965,Y -43.604,Z -178.601,A -90.000,B 90.000,C 0.000} C_DIS
LIN {X 28.381,Y -43.602,Z -178.093,A -90.000,B 90.000,C 0.000} C_DIS
LIN {X 29.602,Y -43.615,Z -176.662,A -90.000,B 90.000,C 0.000} C_DIS
LIN {X 30.192,Y -43.648,Z -175.952,A -90.000,B 90.000,C 0.000} C_DIS
LIN {X 30.532,Y -43.642,Z -175.469,A -90.000,B 90.000,C 0.000} C_DIS
LIN {X 30.863,Y -43.634,Z -175.002,A -90.000,B 90.000,C 0.000} C_DIS
LIN {X 31.081,Y -43.633,Z -174.707,A -90.000,B 90.000,C 0.000} C_DIS
LIN {X 31.546,Y -43.654,Z -174.062,A -90.000,B 90.000,C 0.000} C_DIS
LIN {X 32.224,Y -43.641,Z -172.975,A -90.000,B 90.000,C 0.000} C_DIS
LIN {X 32.409,Y -43.634,Z -172.683,A -90.000,B 90.000,C 0.000} C_DIS
LIN {X 32.464,Y -43.633,Z -172.598,A -90.000,B 90.000,C 0.000} C_DIS
LIN {X 32.732,Y -43.641,Z -172.181,A -90.000,B 90.000,C 0.000} C_DIS
LIN {X 33.770,Y -43.616,Z -170.378,A -90.000,B 90.000,C 0.000} C_DIS
LIN {X 33.894,Y -43.616,Z -170.162,A -90.000,B 90.000,C 0.000} C_DIS
LIN {X 33.993,Y -43.618,Z -169.995,A -90.000,B 90.000,C 0.000} C_DIS
LIN {X 34.740,Y -43.600,Z -168.644,A -90.000,B 90.000,C 0.000} C_DIS
LIN {X 35.045,Y -43.600,Z -168.118,A -90.000,B 90.000,C 0.000} C_DIS
LIN {X 35.265,Y -43.604,Z -167.737,A -90.000,B 90.000,C 0.000} C_DIS
LIN {X 35.504,Y -43.599,Z -167.295,A -90.000,B 90.000,C 0.000} C_DIS
LIN {X 36.493,Y -43.603,Z -165.559,A -90.000,B 90.000,C 0.000} C_DIS
LIN {X 36.970,Y -43.614,Z -164.714,A -90.000,B 90.000,C 0.000} C_DIS
LIN {X 37.384,Y -43.612,Z -163.943,A -90.000,B 90.000,C 0.000} C_DIS
LIN {X 37.638,Y -43.610,Z -163.472,A -90.000,B 90.000,C 0.000} C_DIS
LIN {X 38.115,Y -43.617,Z -162.624,A -90.000,B 90.000,C 0.000} C_DIS
LIN {X 38.634,Y -43.632,Z -161.694,A -90.000,B 90.000,C 0.000} C_DIS
LIN {X 39.983,Y -43.646,Z -159.187,A -90.000,B 90.000,C 0.000} C_DIS
LIN {X 40.055,Y -43.647,Z -159.055,A -90.000,B 90.000,C 0.000} C_DIS
LIN {X 40.374,Y -43.653,Z -158.484,A -90.000,B 90.000,C 0.000} C_DIS
LIN {X 41.055,Y -43.661,Z -157.245,A -90.000,B 90.000,C 0.000} C_DIS
LIN {X 41.378,Y -43.672,Z -156.691,A -90.000,B 90.000,C 0.000} C_DIS
LIN {X 42.260,Y -43.697,Z -155.179,A -90.000,B 90.000,C 0.000} C_DIS
LIN {X 42.920,Y -43.722,Z -154.078,A -90.000,B 90.000,C 0.000} C_DIS
LIN {X 43.378,Y -43.740,Z -153.326,A -90.000,B 90.000,C 0.000} C_DIS
LIN {X 43.921,Y -43.758,Z -152.438,A -90.000,B 90.000,C 0.000} C_DIS
LIN {X 44.208,Y -43.765,Z -151.971,A -90.000,B 90.000,C 0.000} C_DIS
LIN {X 44.398,Y -43.772,Z -151.671,A -90.000,B 90.000,C 0.000} C_DIS
LIN {X 45.149,Y -43.810,Z -150.534,A -90.000,B 90.000,C 0.000} C_DIS
LIN {X 45.392,Y -43.816,Z -150.171,A -90.000,B 90.000,C 0.000} C_DIS
LIN {X 45.916,Y -43.816,Z -149.400,A -90.000,B 90.000,C 0.000} C_DIS
LIN {X 46.553,Y -43.816,Z -148.461,A -90.000,B 90.000,C 0.000} C_DIS
LIN {X 46.634,Y -43.818,Z -148.351,A -90.000,B 90.000,C 0.000} C_DIS
LIN {X 46.756,Y -43.823,Z -148.194,A -90.000,B 90.000,C 0.000} C_DIS
LIN {X 46.818,Y -43.827,Z -148.119,A -90.000,B 90.000,C 0.000} C_DIS
LIN {X 47.618,Y -43.886,Z -147.183,A -90.000,B 90.000,C 0.000} C_DIS
LIN {X 48.834,Y -43.936,Z -145.785,A -90.000,B 90.000,C 0.000} C_DIS
LIN {X 49.603,Y -43.952,Z -144.912,A -90.000,B 90.000,C 0.000} C_DIS
LIN {X 49.868,Y -43.956,Z -144.627,A -90.000,B 90.000,C 0.000} C_DIS
LIN {X 50.405,Y -43.975,Z -144.089,A -90.000,B 90.000,C 0.000} C_DIS
LIN {X 50.709,Y -43.980,Z -143.788,A -90.000,B 90.000,C 0.000} C_DIS
LIN {X 51.082,Y -43.984,Z -143.423,A -90.000,B 90.000,C 0.000} C_DIS
LIN {X 51.773,Y -44.001,Z -142.782,A -90.000,B 90.000,C 0.000} C_DIS
LIN {X 51.928,Y -44.007,Z -142.648,A -90.000,B 90.000,C 0.000} C_DIS
LIN {X 52.869,Y -44.055,Z -141.879,A -90.000,B 90.000,C 0.000} C_DIS
LIN {X 53.347,Y -44.061,Z -141.497,A -90.000,B 90.000,C 0.000} C_DIS
LIN {X 53.670,Y -44.069,Z -141.251,A -90.000,B 90.000,C 0.000} C_DIS
LIN {X 53.812,Y -44.076,Z -141.150,A -90.000,B 90.000,C 0.000} C_DIS
LIN {X 54.677,Y -44.121,Z -140.557,A -90.000,B 90.000,C 0.000} C_DIS
LIN {X 55.178,Y -44.128,Z -140.163,A -90.000,B 90.000,C 0.000} C_DIS
LIN {X 55.397,Y -44.133,Z -139.996,A -90.000,B 90.000,C 0.000} C_DIS
LIN {X 55.501,Y -44.137,Z -139.922,A -90.000,B 90.000,C 0.000} C_DIS
LIN {X 55.707,Y -44.148,Z -139.783,A -90.000,B 90.000,C 0.000} C_DIS
LIN {X 55.813,Y -44.155,Z -139.717,A -90.000,B 90.000,C 0.000} C_DIS
LIN {X 55.884,Y -44.161,Z -139.675,A -90.000,B 90.000,C 0.000} C_DIS
LIN {X 56.093,Y -44.170,Z -139.554,A -90.000,B 90.000,C 0.000} C_DIS
LIN {X 57.273,Y -44.207,Z -138.878,A -90.000,B 90.000,C 0.000} C_DIS
LIN {X 58.657,Y -44.285,Z -138.073,A -90.000,B 90.000,C 0.000} C_DIS
LIN {X 58.886,Y -44.298,Z -137.948,A -90.000,B 90.000,C 0.000} C_DIS
LIN {X 59.002,Y -44.305,Z -137.889,A -90.000,B 90.000,C 0.000} C_DIS
LIN {X 59.292,Y -44.324,Z -137.750,A -90.000,B 90.000,C 0.000} C_DIS
LIN {X 59.438,Y -44.335,Z -137.685,A -90.000,B 90.000,C 0.000} C_DIS
LIN {X 59.934,Y -44.377,Z -137.478,A -90.000,B 90.000,C 0.000} C_DIS
LIN {X 60.553,Y -44.422,Z -137.222,A -90.000,B 90.000,C 0.000} C_DIS
LIN {X 60.757,Y -44.438,Z -137.147,A -90.000,B 90.000,C 0.000} C_DIS
LIN {X 61.993,Y -44.549,Z -136.743,A -90.000,B 90.000,C 0.000} C_DIS
LIN {X 62.781,Y -44.594,Z -136.494,A -90.000,B 90.000,C 0.000} C_DIS
LIN {X 62.975,Y -44.606,Z -136.441,A -90.000,B 90.000,C 0.000} C_DIS
LIN {X 63.116,Y -44.616,Z -136.405,A -90.000,B 90.000,C 0.000} C_DIS
LIN {X 63.251,Y -44.626,Z -136.375,A -90.000,B 90.000,C 0.000} C_DIS
LIN {X 63.549,Y -44.651,Z -136.322,A -90.000,B 90.000,C 0.000} C_DIS
LIN {X 63.647,Y -44.660,Z -136.307,A -90.000,B 90.000,C 0.000} C_DIS
LIN {X 63.785,Y -44.672,Z -136.294,A -90.000,B 90.000,C 0.000} C_DIS
LIN {X 63.906,Y -44.681,Z -136.286,A -90.000,B 90.000,C 0.000} C_DIS
LIN {X 64.113,Y -44.700,Z -136.283,A -90.000,B 90.000,C 0.000} C_DIS
LIN {X 64.424,Y -44.729,Z -136.289,A -90.000,B 90.000,C 0.000} C_DIS
LIN {X 64.805,Y -44.762,Z -136.299,A -90.000,B 90.000,C 0.000} C_DIS
LIN {X 65.763,Y -44.794,Z -136.333,A -90.000,B 90.000,C 0.000} C_DIS
LIN {X 66.078,Y -44.808,Z -136.369,A -90.000,B 90.000,C 0.000} C_DIS
LIN {X 66.556,Y -44.834,Z -136.458,A -90.000,B 90.000,C 0.000} C_DIS
LIN {X 66.726,Y -44.844,Z -136.498,A -90.000,B 90.000,C 0.000} C_DIS
LIN {X 66.825,Y -44.851,Z -136.529,A -90.000,B 90.000,C 0.000} C_DIS
LIN {X 67.456,Y -44.871,Z -136.741,A -90.000,B 90.000,C 0.000} C_DIS
LIN {X 67.665,Y -44.870,Z -136.813,A -90.000,B 90.000,C 0.000} C_DIS
LIN {X 68.238,Y -44.848,Z -137.012,A -90.000,B 90.000,C 0.000} C_DIS
LIN {X 68.334,Y -44.845,Z -137.048,A -90.000,B 90.000,C 0.000} C_DIS
LIN {X 68.519,Y -44.838,Z -137.123,A -90.000,B 90.000,C 0.000} C_DIS
LIN {X 68.655,Y -44.835,Z -137.186,A -90.000,B 90.000,C 0.000} C_DIS
LIN {X 68.968,Y -44.828,Z -137.356,A -90.000,B 90.000,C 0.000} C_DIS
LIN {X 69.075,Y -44.826,Z -137.419,A -90.000,B 90.000,C 0.000} C_DIS
LIN {X 69.170,Y -44.826,Z -137.483,A -90.000,B 90.000,C 0.000} C_DIS
LIN {X 69.377,Y -44.817,Z -137.625,A -90.000,B 90.000,C 0.000} C_DIS
LIN {X 69.470,Y -44.814,Z -137.698,A -90.000,B 90.000,C 0.000} C_DIS
LIN {X 69.692,Y -44.805,Z -137.878,A -90.000,B 90.000,C 0.000} C_DIS
LIN {X 69.780,Y -44.802,Z -137.953,A -90.000,B 90.000,C 0.000} C_DIS
LIN {X 69.926,Y -44.799,Z -138.096,A -90.000,B 90.000,C 0.000} C_DIS
LIN {X 70.443,Y -44.788,Z -138.627,A -90.000,B 90.000,C 0.000} C_DIS
LIN {X 70.557,Y -44.777,Z -138.748,A -90.000,B 90.000,C 0.000} C_DIS
LIN {X 70.671,Y -44.765,Z -138.876,A -90.000,B 90.000,C 0.000} C_DIS
LIN {X 70.866,Y -44.744,Z -139.114,A -90.000,B 90.000,C 0.000} C_DIS
LIN {X 70.980,Y -44.733,Z -139.267,A -90.000,B 90.000,C 0.000} C_DIS
LIN {X 71.024,Y -44.728,Z -139.328,A -90.000,B 90.000,C 0.000} C_DIS
LIN {X 71.119,Y -44.720,Z -139.472,A -90.000,B 90.000,C 0.000} C_DIS
LIN {X 71.173,Y -44.715,Z -139.559,A -90.000,B 90.000,C 0.000} C_DIS
LIN {X 71.622,Y -44.669,Z -140.343,A -90.000,B 90.000,C 0.000} C_DIS
LIN {X 72.207,Y -44.604,Z -141.237,A -90.000,B 90.000,C 0.000} C_DIS
LIN {X 72.275,Y -44.598,Z -141.353,A -90.000,B 90.000,C 0.000} C_DIS
LIN {X 72.436,Y -44.583,Z -141.650,A -90.000,B 90.000,C 0.000} C_DIS
LIN {X 72.510,Y -44.577,Z -141.803,A -90.000,B 90.000,C 0.000} C_DIS
LIN {X 72.995,Y -44.547,Z -142.935,A -90.000,B 90.000,C 0.000} C_DIS
LIN {X 73.173,Y -44.527,Z -143.357,A -90.000,B 90.000,C 0.000} C_DIS
LIN {X 73.205,Y -44.524,Z -143.437,A -90.000,B 90.000,C 0.000} C_DIS
LIN {X 73.311,Y -44.514,Z -143.741,A -90.000,B 90.000,C 0.000} C_DIS
LIN {X 73.342,Y -44.512,Z -143.840,A -90.000,B 90.000,C 0.000} C_DIS
LIN {X 73.476,Y -44.504,Z -144.330,A -90.000,B 90.000,C 0.000} C_DIS
LIN {X 73.641,Y -44.474,Z -144.955,A -90.000,B 90.000,C 0.000} C_DIS
LIN {X 73.679,Y -44.467,Z -145.121,A -90.000,B 90.000,C 0.000} C_DIS
LIN {X 73.709,Y -44.462,Z -145.260,A -90.000,B 90.000,C 0.000} C_DIS
LIN {X 73.728,Y -44.459,Z -145.362,A -90.000,B 90.000,C 0.000} C_DIS
LIN {X 73.775,Y -44.453,Z -145.670,A -90.000,B 90.000,C 0.000} C_DIS
LIN {X 73.917,Y -44.440,Z -146.809,A -90.000,B 90.000,C 0.000} C_DIS
LIN {X 74.156,Y -44.383,Z -148.766,A -90.000,B 90.000,C 0.000} C_DIS
LIN {X 74.231,Y -44.366,Z -149.392,A -90.000,B 90.000,C 0.000} C_DIS
LIN {X 74.265,Y -44.359,Z -149.740,A -90.000,B 90.000,C 0.000} C_DIS
LIN {X 74.278,Y -44.357,Z -149.945,A -90.000,B 90.000,C 0.000} C_DIS
LIN {X 74.302,Y -44.356,Z -150.628,A -90.000,B 90.000,C 0.000} C_DIS
LIN {X 74.355,Y -44.322,Z -152.340,A -90.000,B 90.000,C 0.000} C_DIS
LIN {X 74.408,Y -44.291,Z -153.738,A -90.000,B 90.000,C 0.000} C_DIS
LIN {X 74.410,Y -44.290,Z -153.829,A -90.000,B 90.000,C 0.000} C_DIS
LIN {X 74.409,Y -44.289,Z -154.009,A -90.000,B 90.000,C 0.000} C_DIS
LIN {X 74.406,Y -44.288,Z -154.099,A -90.000,B 90.000,C 0.000} C_DIS
LIN {X 74.385,Y -44.290,Z -154.532,A -90.000,B 90.000,C 0.000} C_DIS
LIN {X 74.204,Y -44.242,Z -157.910,A -90.000,B 90.000,C 0.000} C_DIS
LIN {X 74.172,Y -44.238,Z -158.297,A -90.000,B 90.000,C 0.000} C_DIS
LIN {X 74.146,Y -44.239,Z -158.504,A -90.000,B 90.000,C 0.000} C_DIS
LIN {X 74.136,Y -44.238,Z -158.565,A -90.000,B 90.000,C 0.000} C_DIS
LIN {X 73.996,Y -44.229,Z -159.458,A -90.000,B 90.000,C 0.000} C_DIS
LIN {X 73.457,Y -44.223,Z -162.352,A -90.000,B 90.000,C 0.000} C_DIS
LIN {X 73.433,Y -44.221,Z -162.456,A -90.000,B 90.000,C 0.000} C_DIS
LIN {X 73.382,Y -44.219,Z -162.653,A -90.000,B 90.000,C 0.000} C_DIS
LIN {X 72.465,Y -44.216,Z -165.833,A -90.000,B 90.000,C 0.000} C_DIS
LIN {X 72.322,Y -44.207,Z -166.323,A -90.000,B 90.000,C 0.000} C_DIS
LIN {X 72.270,Y -44.205,Z -166.487,A -90.000,B 90.000,C 0.000} C_DIS
LIN {X 72.235,Y -44.205,Z -166.591,A -90.000,B 90.000,C 0.000} C_DIS
LIN {X 72.159,Y -44.205,Z -166.806,A -90.000,B 90.000,C 0.000} C_DIS
LIN {X 71.199,Y -44.200,Z -169.543,A -90.000,B 90.000,C 0.000} C_DIS
LIN {X 71.077,Y -44.199,Z -169.891,A -90.000,B 90.000,C 0.000} C_DIS
LIN {X 70.541,Y -44.197,Z -171.356,A -90.000,B 90.000,C 0.000} C_DIS
LIN {X 70.159,Y -44.201,Z -172.353,A -90.000,B 90.000,C 0.000} C_DIS
LIN {X 69.912,Y -44.211,Z -173.008,A -90.000,B 90.000,C 0.000} C_DIS
LIN {X 69.180,Y -44.213,Z -175.215,A -90.000,B 90.000,C 0.000} C_DIS
LIN {X 69.066,Y -44.223,Z -175.567,A -90.000,B 90.000,C 0.000} C_DIS
LIN {X 68.688,Y -44.214,Z -177.417,A -90.000,B 90.000,C 0.000} C_DIS
LIN {X 68.545,Y -44.215,Z -178.059,A -90.000,B 90.000,C 0.000} C_DIS
LIN {X 68.282,Y -44.215,Z -179.891,A -90.000,B 90.000,C 0.000} C_DIS
LIN {X 68.191,Y -44.209,Z -180.508,A -90.000,B 90.000,C 0.000} C_DIS
LIN {X 68.172,Y -44.204,Z -180.725,A -90.000,B 90.000,C 0.000} C_DIS
LIN {X 67.981,Y -44.174,Z -182.827,A -90.000,B 90.000,C 0.000} C_DIS
LIN {X 67.928,Y -44.152,Z -183.718,A -90.000,B 90.000,C 0.000} C_DIS
LIN {X 67.772,Y -44.110,Z -186.062,A -90.000,B 90.000,C 0.000} C_DIS
LIN {X 67.704,Y -44.088,Z -187.029,A -90.000,B 90.000,C 0.000} C_DIS
LIN {X 67.642,Y -44.072,Z -187.878,A -90.000,B 90.000,C 0.000} C_DIS
LIN {X 67.612,Y -44.066,Z -188.241,A -90.000,B 90.000,C 0.000} C_DIS
LIN {X 67.578,Y -44.061,Z -188.562,A -90.000,B 90.000,C 0.000} C_DIS
LIN {X 67.379,Y -44.020,Z -190.393,A -90.000,B 90.000,C 0.000} C_DIS
LIN {X 67.318,Y -44.010,Z -190.959,A -90.000,B 90.000,C 0.000} C_DIS
LIN {X 67.294,Y -44.008,Z -191.127,A -90.000,B 90.000,C 0.000} C_DIS
LIN {X 67.263,Y -44.007,Z -191.322,A -90.000,B 90.000,C 0.000} C_DIS
LIN {X 66.808,Y -43.954,Z -194.042,A -90.000,B 90.000,C 0.000} C_DIS
LIN {X 66.774,Y -43.953,Z -194.216,A -90.000,B 90.000,C 0.000} C_DIS
LIN {X 66.409,Y -43.928,Z -195.792,A -90.000,B 90.000,C 0.000} C_DIS
LIN {X 65.997,Y -43.908,Z -197.500,A -90.000,B 90.000,C 0.000} C_DIS
LIN {X 65.962,Y -43.905,Z -197.639,A -90.000,B 90.000,C 0.000} C_DIS
LIN {X 65.897,Y -43.901,Z -197.872,A -90.000,B 90.000,C 0.000} C_DIS
LIN {X 65.419,Y -43.885,Z -199.474,A -90.000,B 90.000,C 0.000} C_DIS
LIN {X 65.215,Y -43.877,Z -200.158,A -90.000,B 90.000,C 0.000} C_DIS
LIN {X 64.793,Y -43.873,Z -201.479,A -90.000,B 90.000,C 0.000} C_DIS
LIN {X 64.682,Y -43.869,Z -201.817,A -90.000,B 90.000,C 0.000} C_DIS
LIN {X 63.502,Y -43.863,Z -205.165,A -90.000,B 90.000,C 0.000} C_DIS
LIN {X 63.200,Y -43.856,Z -206.013,A -90.000,B 90.000,C 0.000} C_DIS
LIN {X 63.039,Y -43.849,Z -206.458,A -90.000,B 90.000,C 0.000} C_DIS
LIN {X 61.367,Y -43.817,Z -210.881,A -90.000,B 90.000,C 0.000} C_DIS
LIN {X 61.239,Y -43.812,Z -211.217,A -90.000,B 90.000,C 0.000} C_DIS
LIN {X 59.377,Y -43.777,Z -215.933,A -90.000,B 90.000,C 0.000} C_DIS
LIN {X 59.258,Y -43.774,Z -216.232,A -90.000,B 90.000,C 0.000} C_DIS
LIN {X 57.513,Y -43.737,Z -220.510,A -90.000,B 90.000,C 0.000} C_DIS
LIN {X 57.242,Y -43.730,Z -221.172,A -90.000,B 90.000,C 0.000} C_DIS
LIN {X 57.116,Y -43.724,Z -221.473,A -90.000,B 90.000,C 0.000} C_DIS
LIN {X 54.882,Y -43.692,Z -226.445,A -90.000,B 90.000,C 0.000} C_DIS
LIN {X 54.693,Y -43.681,Z -226.854,A -90.000,B 90.000,C 0.000} C_DIS
LIN {X 54.640,Y -43.679,Z -226.959,A -90.000,B 90.000,C 0.000} C_DIS
LIN {X 53.122,Y -43.682,Z -229.862,A -90.000,B 90.000,C 0.000} C_DIS
LIN {X 52.553,Y -43.681,Z -230.970,A -90.000,B 90.000,C 0.000} C_DIS
LIN {X 52.169,Y -43.681,Z -231.718,A -90.000,B 90.000,C 0.000} C_DIS
LIN {X 51.927,Y -43.669,Z -232.177,A -90.000,B 90.000,C 0.000} C_DIS
LIN {X 51.845,Y -43.664,Z -232.326,A -90.000,B 90.000,C 0.000} C_DIS
LIN {X 51.664,Y -43.661,Z -232.637,A -90.000,B 90.000,C 0.000} C_DIS
LIN {X 51.622,Y -43.661,Z -232.706,A -90.000,B 90.000,C 0.000} C_DIS
LIN {X 49.770,Y -43.699,Z -235.639,A -90.000,B 90.000,C 0.000} C_DIS
LIN {X 49.528,Y -43.701,Z -236.033,A -90.000,B 90.000,C 0.000} C_DIS
LIN {X 48.817,Y -43.715,Z -237.201,A -90.000,B 90.000,C 0.000} C_DIS
LIN {X 48.436,Y -43.691,Z -237.803,A -90.000,B 90.000,C 0.000} C_DIS
LIN {X 48.358,Y -43.688,Z -237.921,A -90.000,B 90.000,C 0.000} C_DIS
LIN {X 48.288,Y -43.687,Z -238.021,A -90.000,B 90.000,C 0.000} C_DIS
LIN {X 48.171,Y -43.688,Z -238.178,A -90.000,B 90.000,C 0.000} C_DIS
LIN {X 45.500,Y -43.794,Z -241.554,A -90.000,B 90.000,C 0.000} C_DIS
LIN {X 45.414,Y -43.799,Z -241.664,A -90.000,B 90.000,C 0.000} C_DIS
LIN {X 45.106,Y -43.812,Z -242.074,A -90.000,B 90.000,C 0.000} C_DIS
LIN {X 45.042,Y -43.815,Z -242.159,A -90.000,B 90.000,C 0.000} C_DIS
LIN {X 44.352,Y -43.799,Z -243.048,A -90.000,B 90.000,C 0.000} C_DIS
LIN {X 44.186,Y -43.799,Z -243.249,A -90.000,B 90.000,C 0.000} C_DIS
LIN {X 44.058,Y -43.801,Z -243.400,A -90.000,B 90.000,C 0.000} C_DIS
LIN {X 43.913,Y -43.806,Z -243.561,A -90.000,B 90.000,C 0.000} C_DIS
LIN {X 43.913,Y -60.000,Z -243.561,A -90.000,B 90.000,C 0.000} C_DIS
LIN {X -31.481,Y -60.000,Z -224.619,A -90.000,B 90.000,C 0.000} C_DIS
LIN {X -31.481,Y -43.308,Z -224.619,A -90.000,B 90.000,C 0.000} C_DIS
LIN {X -31.198,Y -43.332,Z -224.571,A -90.000,B 90.000,C 0.000} C_DIS
LIN {X -30.977,Y -43.353,Z -224.541,A -90.000,B 90.000,C 0.000} C_DIS
LIN {X -30.295,Y -43.422,Z -224.458,A -90.000,B 90.000,C 0.000} C_DIS
LIN {X -29.742,Y -43.475,Z -224.394,A -90.000,B 90.000,C 0.000} C_DIS
LIN {X -27.960,Y -43.670,Z -224.245,A -90.000,B 90.000,C 0.000} C_DIS
LIN {X -27.759,Y -43.684,Z -224.231,A -90.000,B 90.000,C 0.000} C_DIS
LIN {X -27.348,Y -43.709,Z -224.204,A -90.000,B 90.000,C 0.000} C_DIS
LIN {X -26.319,Y -43.762,Z -224.103,A -90.000,B 90.000,C 0.000} C_DIS
LIN {X -25.709,Y -43.793,Z -224.058,A -90.000,B 90.000,C 0.000} C_DIS
LIN {X -25.245,Y -43.823,Z -224.042,A -90.000,B 90.000,C 0.000} C_DIS
LIN {X -25.140,Y -43.831,Z -224.041,A -90.000,B 90.000,C 0.000} C_DIS
LIN {X -24.837,Y -43.855,Z -224.046,A -90.000,B 90.000,C 0.000} C_DIS
LIN {X -24.637,Y -43.873,Z -224.056,A -90.000,B 90.000,C 0.000} C_DIS
LIN {X -24.114,Y -43.921,Z -224.087,A -90.000,B 90.000,C 0.000} C_DIS
LIN {X -24.009,Y -43.931,Z -224.096,A -90.000,B 90.000,C 0.000} C_DIS
LIN {X -23.666,Y -43.968,Z -224.134,A -90.000,B 90.000,C 0.000} C_DIS
LIN {X -23.369,Y -44.004,Z -224.181,A -90.000,B 90.000,C 0.000} C_DIS
LIN {X -23.046,Y -44.046,Z -224.237,A -90.000,B 90.000,C 0.000} C_DIS
LIN {X -22.724,Y -44.090,Z -224.293,A -90.000,B 90.000,C 0.000} C_DIS
LIN {X -22.591,Y -44.104,Z -224.318,A -90.000,B 90.000,C 0.000} C_DIS
LIN {X -21.126,Y -44.203,Z -224.598,A -90.000,B 90.000,C 0.000} C_DIS
LIN {X -19.698,Y -44.309,Z -224.918,A -90.000,B 90.000,C 0.000} C_DIS
LIN {X -19.478,Y -44.327,Z -224.975,A -90.000,B 90.000,C 0.000} C_DIS
LIN {X -19.167,Y -44.354,Z -225.069,A -90.000,B 90.000,C 0.000} C_DIS
LIN {X -18.889,Y -44.376,Z -225.162,A -90.000,B 90.000,C 0.000} C_DIS
LIN {X -18.758,Y -44.387,Z -225.211,A -90.000,B 90.000,C 0.000} C_DIS
LIN {X -18.634,Y -44.394,Z -225.263,A -90.000,B 90.000,C 0.000} C_DIS
LIN {X -18.410,Y -44.403,Z -225.361,A -90.000,B 90.000,C 0.000} C_DIS
LIN {X -18.231,Y -44.411,Z -225.448,A -90.000,B 90.000,C 0.000} C_DIS
LIN {X -18.078,Y -44.419,Z -225.531,A -90.000,B 90.000,C 0.000} C_DIS
LIN {X -17.787,Y -44.437,Z -225.701,A -90.000,B 90.000,C 0.000} C_DIS
LIN {X -17.541,Y -44.454,Z -225.860,A -90.000,B 90.000,C 0.000} C_DIS
LIN {X -17.187,Y -44.480,Z -226.103,A -90.000,B 90.000,C 0.000} C_DIS
LIN {X -16.258,Y -44.551,Z -226.748,A -90.000,B 90.000,C 0.000} C_DIS
LIN {X -16.109,Y -44.557,Z -226.853,A -90.000,B 90.000,C 0.000} C_DIS
LIN {X -15.985,Y -44.558,Z -226.945,A -90.000,B 90.000,C 0.000} C_DIS
LIN {X -14.888,Y -44.559,Z -227.772,A -90.000,B 90.000,C 0.000} C_DIS
LIN {X -14.736,Y -44.560,Z -227.896,A -90.000,B 90.000,C 0.000} C_DIS
LIN {X -14.462,Y -44.564,Z -228.135,A -90.000,B 90.000,C 0.000} C_DIS
LIN {X -14.316,Y -44.568,Z -228.274,A -90.000,B 90.000,C 0.000} C_DIS
LIN {X -14.226,Y -44.570,Z -228.365,A -90.000,B 90.000,C 0.000} C_DIS
LIN {X -14.031,Y -44.577,Z -228.577,A -90.000,B 90.000,C 0.000} C_DIS
LIN {X -13.923,Y -44.581,Z -228.702,A -90.000,B 90.000,C 0.000} C_DIS
LIN {X -13.817,Y -44.581,Z -228.830,A -90.000,B 90.000,C 0.000} C_DIS
LIN {X -13.765,Y -44.579,Z -228.894,A -90.000,B 90.000,C 0.000} C_DIS
LIN {X -13.665,Y -44.576,Z -229.025,A -90.000,B 90.000,C 0.000} C_DIS
LIN {X -13.498,Y -44.570,Z -229.256,A -90.000,B 90.000,C 0.000} C_DIS
LIN {X -13.357,Y -44.567,Z -229.473,A -90.000,B 90.000,C 0.000} C_DIS
LIN {X -12.770,Y -44.555,Z -230.443,A -90.000,B 90.000,C 0.000} C_DIS
LIN {X -12.366,Y -44.552,Z -231.110,A -90.000,B 90.000,C 0.000} C_DIS
LIN {X -11.836,Y -44.532,Z -232.011,A -90.000,B 90.000,C 0.000} C_DIS
LIN {X -11.665,Y -44.526,Z -232.328,A -90.000,B 90.000,C 0.000} C_DIS
LIN {X -11.567,Y -44.523,Z -232.528,A -90.000,B 90.000,C 0.000} C_DIS
LIN {X -11.065,Y -44.515,Z -233.650,A -90.000,B 90.000,C 0.000} C_DIS
LIN {X -10.751,Y -44.528,Z -234.347,A -90.000,B 90.000,C 0.000} C_DIS
LIN {X -10.501,Y -44.546,Z -234.901,A -90.000,B 90.000,C 0.000} C_DIS
LIN {X -9.909,Y -44.562,Z -235.872,A -90.000,B 90.000,C 0.000} C_DIS
LIN {X -9.726,Y -44.566,Z -236.146,A -90.000,B 90.000,C 0.000} C_DIS
LIN {X -9.495,Y -44.566,Z -236.316,A -90.000,B 90.000,C 0.000} C_DIS
LIN {X -9.157,Y -44.558,Z -236.374,A -90.000,B 90.000,C 0.000} C_DIS
LIN {X -8.944,Y -44.549,Z -236.376,A -90.000,B 90.000,C 0.000} C_DIS
LIN {X -8.097,Y -44.481,Z -236.083,A -90.000,B 90.000,C 0.000} C_DIS
LIN {X -6.366,Y -44.371,Z -235.478,A -90.000,B 90.000,C 0.000} C_DIS
LIN {X -4.930,Y -44.323,Z -234.970,A -90.000,B 90.000,C 0.000} C_DIS
LIN {X -4.401,Y -44.319,Z -234.781,A -90.000,B 90.000,C 0.000} C_DIS
LIN {X -3.145,Y -44.222,Z -233.732,A -90.000,B 90.000,C 0.000} C_DIS
LIN {X -2.844,Y -44.210,Z -233.477,A -90.000,B 90.000,C 0.000} C_DIS
LIN {X -2.501,Y -44.198,Z -233.189,A -90.000,B 90.000,C 0.000} C_DIS
LIN {X -1.550,Y -44.181,Z -232.416,A -90.000,B 90.000,C 0.000} C_DIS
LIN {X 0.361,Y -44.053,Z -230.189,A -90.000,B 90.000,C 0.000} C_DIS
LIN {X 1.252,Y -44.021,Z -229.143,A -90.000,B 90.000,C 0.000} C_DIS
LIN {X 1.441,Y -44.011,Z -228.869,A -90.000,B 90.000,C 0.000} C_DIS
LIN {X 3.730,Y -43.889,Z -225.519,A -90.000,B 90.000,C 0.000} C_DIS
LIN {X 4.147,Y -43.878,Z -224.905,A -90.000,B 90.000,C 0.000} C_DIS
LIN {X 4.502,Y -43.877,Z -224.392,A -90.000,B 90.000,C 0.000} C_DIS
LIN {X 4.638,Y -43.878,Z -224.193,A -90.000,B 90.000,C 0.000} C_DIS
LIN {X 5.899,Y -43.873,Z -222.116,A -90.000,B 90.000,C 0.000} C_DIS
LIN {X 6.873,Y -43.870,Z -220.509,A -90.000,B 90.000,C 0.000} C_DIS
LIN {X 7.218,Y -43.874,Z -219.938,A -90.000,B 90.000,C 0.000} C_DIS
LIN {X 8.205,Y -43.876,Z -218.182,A -90.000,B 90.000,C 0.000} C_DIS
LIN {X 8.771,Y -43.887,Z -217.172,A -90.000,B 90.000,C 0.000} C_DIS
LIN {X 9.340,Y -43.900,Z -216.188,A -90.000,B 90.000,C 0.000} C_DIS
LIN {X 9.752,Y -43.916,Z -215.472,A -90.000,B 90.000,C 0.000} C_DIS
LIN {X 10.602,Y -43.939,Z -213.838,A -90.000,B 90.000,C 0.000} C_DIS
LIN {X 10.978,Y -43.947,Z -213.089,A -90.000,B 90.000,C 0.000} C_DIS
LIN {X 11.962,Y -43.984,Z -211.120,A -90.000,B 90.000,C 0.000} C_DIS
LIN {X 12.184,Y -43.992,Z -210.651,A -90.000,B 90.000,C 0.000} C_DIS
LIN {X 12.289,Y -43.995,Z -210.400,A -90.000,B 90.000,C 0.000} C_DIS
LIN {X 12.653,Y -44.010,Z -209.527,A -90.000,B 90.000,C 0.000} C_DIS
LIN {X 13.468,Y -44.042,Z -207.559,A -90.000,B 90.000,C 0.000} C_DIS
LIN {X 13.695,Y -44.051,Z -206.986,A -90.000,B 90.000,C 0.000} C_DIS
LIN {X 14.397,Y -44.065,Z -204.944,A -90.000,B 90.000,C 0.000} C_DIS
LIN {X 14.729,Y -44.059,Z -203.838,A -90.000,B 90.000,C 0.000} C_DIS
LIN {X 14.964,Y -44.050,Z -203.056,A -90.000,B 90.000,C 0.000} C_DIS
LIN {X 15.028,Y -44.046,Z -202.815,A -90.000,B 90.000,C 0.000} C_DIS
LIN {X 15.144,Y -44.026,Z -202.214,A -90.000,B 90.000,C 0.000} C_DIS
LIN {X 15.812,Y -43.925,Z -198.993,A -90.000,B 90.000,C 0.000} C_DIS
LIN {X 15.852,Y -43.918,Z -198.794,A -90.000,B 90.000,C 0.000} C_DIS
LIN {X 16.025,Y -43.869,Z -197.960,A -90.000,B 90.000,C 0.000} C_DIS
LIN {X 16.428,Y -43.732,Z -196.060,A -90.000,B 90.000,C 0.000} C_DIS
LIN {X 16.467,Y -43.722,Z -195.904,A -90.000,B 90.000,C 0.000} C_DIS
LIN {X 16.854,Y -43.640,Z -194.489,A -90.000,B 90.000,C 0.000} C_DIS
LIN {X 16.906,Y -43.632,Z -194.319,A -90.000,B 90.000,C 0.000} C_DIS
LIN {X 17.026,Y -43.615,Z -193.952,A -90.000,B 90.000,C 0.000} C_DIS
LIN {X 17.072,Y -43.609,Z -193.825,A -90.000,B 90.000,C 0.000} C_DIS
LIN {X 17.217,Y -43.596,Z -193.415,A -90.000,B 90.000,C 0.000} C_DIS
LIN {X 17.423,Y -43.564,Z -192.850,A -90.000,B 90.000,C 0.000} C_DIS
LIN {X 17.540,Y -43.542,Z -192.505,A -90.000,B 90.000,C 0.000} C_DIS
LIN {X 18.307,Y -43.360,Z -190.275,A -90.000,B 90.000,C 0.000} C_DIS
LIN {X 18.404,Y -43.342,Z -190.021,A -90.000,B 90.000,C 0.000} C_DIS
LIN {X 18.458,Y -43.335,Z -189.890,A -90.000,B 90.000,C 0.000} C_DIS
LIN {X 18.647,Y -43.314,Z -189.464,A -90.000,B 90.000,C 0.000} C_DIS
LIN {X 18.708,Y -43.308,Z -189.335,A -90.000,B 90.000,C 0.000} C_DIS
LIN {X 18.708,Y -60.000,Z -189.335,A -90.000,B 90.000,C 0.000} C_DIS
LIN {X -24.634,Y -60.000,Z -222.132,A -90.000,B 90.000,C 0.000} C_DIS
LIN {X -24.634,Y -43.308,Z -222.132,A -90.000,B 90.000,C 0.000} C_DIS
LIN {X -23.951,Y -43.379,Z -222.169,A -90.000,B 90.000,C 0.000} C_DIS
LIN {X -23.725,Y -43.405,Z -222.188,A -90.000,B 90.000,C 0.000} C_DIS
LIN {X -23.397,Y -43.444,Z -222.223,A -90.000,B 90.000,C 0.000} C_DIS
LIN {X -23.254,Y -43.462,Z -222.243,A -90.000,B 90.000,C 0.000} C_DIS
LIN {X -22.972,Y -43.499,Z -222.287,A -90.000,B 90.000,C 0.000} C_DIS
LIN {X -20.732,Y -43.806,Z -222.677,A -90.000,B 90.000,C 0.000} C_DIS
LIN {X -20.674,Y -43.814,Z -222.688,A -90.000,B 90.000,C 0.000} C_DIS
LIN {X -20.545,Y -43.828,Z -222.716,A -90.000,B 90.000,C 0.000} C_DIS
LIN {X -19.179,Y -43.930,Z -223.024,A -90.000,B 90.000,C 0.000} C_DIS
LIN {X -18.881,Y -43.955,Z -223.103,A -90.000,B 90.000,C 0.000} C_DIS
LIN {X -18.516,Y -43.988,Z -223.213,A -90.000,B 90.000,C 0.000} C_DIS
LIN {X -18.179,Y -44.021,Z -223.326,A -90.000,B 90.000,C 0.000} C_DIS
LIN {X -17.977,Y -44.042,Z -223.402,A -90.000,B 90.000,C 0.000} C_DIS
LIN {X -17.605,Y -44.085,Z -223.558,A -90.000,B 90.000,C 0.000} C_DIS
LIN {X -17.397,Y -44.110,Z -223.655,A -90.000,B 90.000,C 0.000} C_DIS
LIN {X -17.281,Y -44.122,Z -223.713,A -90.000,B 90.000,C 0.000} C_DIS
LIN {X -17.065,Y -44.147,Z -223.828,A -90.000,B 90.000,C 0.000} C_DIS
LIN {X -16.936,Y -44.159,Z -223.903,A -90.000,B 90.000,C 0.000} C_DIS
LIN {X -16.776,Y -44.169,Z -223.997,A -90.000,B 90.000,C 0.000} C_DIS
LIN {X -16.699,Y -44.174,Z -224.044,A -90.000,B 90.000,C 0.000} C_DIS
LIN {X -16.407,Y -44.194,Z -224.234,A -90.000,B 90.000,C 0.000} C_DIS
LIN {X -15.548,Y -44.259,Z -224.827,A -90.000,B 90.000,C 0.000} C_DIS
LIN {X -14.921,Y -44.308,Z -225.264,A -90.000,B 90.000,C 0.000} C_DIS
LIN {X -14.644,Y -44.330,Z -225.467,A -90.000,B 90.000,C 0.000} C_DIS
LIN {X -14.514,Y -44.335,Z -225.564,A -90.000,B 90.000,C 0.000} C_DIS
LIN {X -13.668,Y -44.337,Z -226.203,A -90.000,B 90.000,C 0.000} C_DIS
LIN {X -13.427,Y -44.340,Z -226.400,A -90.000,B 90.000,C 0.000} C_DIS
LIN {X -13.153,Y -44.344,Z -226.639,A -90.000,B 90.000,C 0.000} C_DIS
LIN {X -13.017,Y -44.347,Z -226.766,A -90.000,B 90.000,C 0.000} C_DIS
LIN {X -12.880,Y -44.351,Z -226.899,A -90.000,B 90.000,C 0.000} C_DIS
LIN {X -12.759,Y -44.354,Z -227.023,A -90.000,B 90.000,C 0.000} C_DIS
LIN {X -12.510,Y -44.363,Z -227.296,A -90.000,B 90.000,C 0.000} C_DIS
LIN {X -12.385,Y -44.367,Z -227.441,A -90.000,B 90.000,C 0.000} C_DIS
LIN {X -12.300,Y -44.367,Z -227.544,A -90.000,B 90.000,C 0.000} C_DIS
LIN {X -12.189,Y -44.363,Z -227.682,A -90.000,B 90.000,C 0.000} C_DIS
LIN {X -12.045,Y -44.358,Z -227.872,A -90.000,B 90.000,C 0.000} C_DIS
LIN {X -11.839,Y -44.351,Z -228.161,A -90.000,B 90.000,C 0.000} C_DIS
LIN {X -11.653,Y -44.348,Z -228.447,A -90.000,B 90.000,C 0.000} C_DIS
LIN {X -10.850,Y -44.341,Z -229.773,A -90.000,B 90.000,C 0.000} C_DIS
LIN {X -10.654,Y -44.334,Z -230.099,A -90.000,B 90.000,C 0.000} C_DIS
LIN {X -10.089,Y -44.312,Z -231.062,A -90.000,B 90.000,C 0.000} C_DIS
LIN {X -9.918,Y -44.310,Z -231.378,A -90.000,B 90.000,C 0.000} C_DIS
LIN {X -9.882,Y -44.309,Z -231.449,A -90.000,B 90.000,C 0.000} C_DIS
LIN {X -9.751,Y -44.309,Z -231.717,A -90.000,B 90.000,C 0.000} C_DIS
LIN {X -9.500,Y -44.311,Z -232.277,A -90.000,B 90.000,C 0.000} C_DIS
LIN {X -8.736,Y -44.342,Z -233.973,A -90.000,B 90.000,C 0.000} C_DIS
LIN {X -8.627,Y -44.343,Z -234.153,A -90.000,B 90.000,C 0.000} C_DIS
LIN {X -8.514,Y -44.332,Z -234.114,A -90.000,B 90.000,C 0.000} C_DIS
LIN {X -7.413,Y -44.242,Z -233.731,A -90.000,B 90.000,C 0.000} C_DIS
LIN {X -5.689,Y -44.132,Z -233.127,A -90.000,B 90.000,C 0.000} C_DIS
LIN {X -5.411,Y -44.122,Z -233.029,A -90.000,B 90.000,C 0.000} C_DIS
LIN {X -4.128,Y -44.016,Z -231.957,A -90.000,B 90.000,C 0.000} C_DIS
LIN {X -3.749,Y -43.994,Z -231.639,A -90.000,B 90.000,C 0.000} C_DIS
LIN {X -2.946,Y -43.949,Z -230.991,A -90.000,B 90.000,C 0.000} C_DIS
LIN {X -2.238,Y -43.888,Z -230.168,A -90.000,B 90.000,C 0.000} C_DIS
LIN {X -0.477,Y -43.779,Z -228.112,A -90.000,B 90.000,C 0.000} C_DIS
LIN {X -0.328,Y -43.774,Z -227.937,A -90.000,B 90.000,C 0.000} C_DIS
LIN {X 1.534,Y -43.667,Z -225.216,A -90.000,B 90.000,C 0.000} C_DIS
LIN {X 2.350,Y -43.637,Z -224.018,A -90.000,B 90.000,C 0.000} C_DIS
LIN {X 2.523,Y -43.635,Z -223.763,A -90.000,B 90.000,C 0.000} C_DIS
LIN {X 2.970,Y -43.631,Z -223.115,A -90.000,B 90.000,C 0.000} C_DIS
LIN {X 4.117,Y -43.605,Z -221.231,A -90.000,B 90.000,C 0.000} C_DIS
LIN {X 5.052,Y -43.600,Z -219.690,A -90.000,B 90.000,C 0.000} C_DIS
LIN {X 5.178,Y -43.600,Z -219.482,A -90.000,B 90.000,C 0.000} C_DIS
LIN {X 5.523,Y -43.601,Z -218.911,A -90.000,B 90.000,C 0.000} C_DIS
LIN {X 5.681,Y -43.602,Z -218.630,A -90.000,B 90.000,C 0.000} C_DIS
LIN {X 7.055,Y -43.628,Z -216.177,A -90.000,B 90.000,C 0.000} C_DIS
LIN {X 7.777,Y -43.645,Z -214.928,A -90.000,B 90.000,C 0.000} C_DIS
LIN {X 8.014,Y -43.652,Z -214.516,A -90.000,B 90.000,C 0.000} C_DIS
LIN {X 8.848,Y -43.669,Z -212.915,A -90.000,B 90.000,C 0.000} C_DIS
LIN {X 9.676,Y -43.683,Z -211.266,A -90.000,B 90.000,C 0.000} C_DIS
LIN {X 10.194,Y -43.702,Z -210.229,A -90.000,B 90.000,C 0.000} C_DIS
LIN {X 10.376,Y -43.707,Z -209.842,A -90.000,B 90.000,C 0.000} C_DIS
LIN {X 10.830,Y -43.712,Z -208.761,A -90.000,B 90.000,C 0.000} C_DIS
LIN {X 11.643,Y -43.720,Z -206.807,A -90.000,B 90.000,C 0.000} C_DIS
LIN {X 11.845,Y -43.721,Z -206.300,A -90.000,B 90.000,C 0.000} C_DIS
LIN {X 12.525,Y -43.703,Z -204.342,A -90.000,B 90.000,C 0.000} C_DIS
LIN {X 12.756,Y -43.691,Z -203.574,A -90.000,B 90.000,C 0.000} C_DIS
LIN {X 13.083,Y -43.662,Z -202.493,A -90.000,B 90.000,C 0.000} C_DIS
LIN {X 13.112,Y -43.658,Z -202.386,A -90.000,B 90.000,C 0.000} C_DIS
LIN {X 13.232,Y -43.624,Z -201.784,A -90.000,B 90.000,C 0.000} C_DIS
LIN {X 13.947,Y -43.432,Z -198.428,A -90.000,B 90.000,C 0.000} C_DIS
LIN {X 14.108,Y -43.386,Z -197.652,A -90.000,B 90.000,C 0.000} C_DIS
LIN {X 14.297,Y -43.308,Z -196.776,A -90.000,B 90.000,C 0.000} C_DIS
LIN {X 14.297,Y -60.000,Z -196.776,A -90.000,B 90.000,C 0.000} C_DIS
LIN {X -20.295,Y -60.000,Z -220.790,A -90.000,B 90.000,C 0.000} C_DIS
LIN {X -20.295,Y -43.308,Z -220.790,A -90.000,B 90.000,C 0.000} C_DIS
LIN {X -19.206,Y -43.468,Z -221.015,A -90.000,B 90.000,C 0.000} C_DIS
LIN {X -18.667,Y -43.547,Z -221.129,A -90.000,B 90.000,C 0.000} C_DIS
LIN {X -18.554,Y -43.560,Z -221.158,A -90.000,B 90.000,C 0.000} C_DIS
LIN {X -18.280,Y -43.583,Z -221.232,A -90.000,B 90.000,C 0.000} C_DIS
LIN {X -17.860,Y -43.621,Z -221.360,A -90.000,B 90.000,C 0.000} C_DIS
LIN {X -17.456,Y -43.661,Z -221.497,A -90.000,B 90.000,C 0.000} C_DIS
LIN {X -17.180,Y -43.690,Z -221.601,A -90.000,B 90.000,C 0.000} C_DIS
LIN {X -16.808,Y -43.733,Z -221.758,A -90.000,B 90.000,C 0.000} C_DIS
LIN {X -16.524,Y -43.768,Z -221.889,A -90.000,B 90.000,C 0.000} C_DIS
LIN {X -16.320,Y -43.796,Z -221.989,A -90.000,B 90.000,C 0.000} C_DIS
LIN {X -16.052,Y -43.834,Z -222.132,A -90.000,B 90.000,C 0.000} C_DIS
LIN {X -15.774,Y -43.876,Z -222.290,A -90.000,B 90.000,C 0.000} C_DIS
LIN {X -15.607,Y -43.902,Z -222.391,A -90.000,B 90.000,C 0.000} C_DIS
LIN {X -15.413,Y -43.932,Z -222.514,A -90.000,B 90.000,C 0.000} C_DIS
LIN {X -15.266,Y -43.944,Z -222.610,A -90.000,B 90.000,C 0.000} C_DIS
LIN {X -14.407,Y -44.012,Z -223.203,A -90.000,B 90.000,C 0.000} C_DIS
LIN {X -13.734,Y -44.065,Z -223.673,A -90.000,B 90.000,C 0.000} C_DIS
LIN {X -13.290,Y -44.104,Z -224.000,A -90.000,B 90.000,C 0.000} C_DIS
LIN {X -13.107,Y -44.121,Z -224.135,A -90.000,B 90.000,C 0.000} C_DIS
LIN {X -12.971,Y -44.126,Z -224.237,A -90.000,B 90.000,C 0.000} C_DIS
LIN {X -12.470,Y -44.129,Z -224.615,A -90.000,B 90.000,C 0.000} C_DIS
LIN {X -12.167,Y -44.132,Z -224.861,A -90.000,B 90.000,C 0.000} C_DIS
LIN {X -11.794,Y -44.138,Z -225.186,A -90.000,B 90.000,C 0.000} C_DIS
LIN {X -11.629,Y -44.142,Z -225.340,A -90.000,B 90.000,C 0.000} C_DIS
LIN {X -11.450,Y -44.146,Z -225.515,A -90.000,B 90.000,C 0.000} C_DIS
LIN {X -11.285,Y -44.150,Z -225.687,A -90.000,B 90.000,C 0.000} C_DIS
LIN {X -11.196,Y -44.153,Z -225.785,A -90.000,B 90.000,C 0.000} C_DIS
LIN {X -10.999,Y -44.162,Z -226.001,A -90.000,B 90.000,C 0.000} C_DIS
LIN {X -10.846,Y -44.167,Z -226.179,A -90.000,B 90.000,C 0.000} C_DIS
LIN {X -10.636,Y -44.160,Z -226.438,A -90.000,B 90.000,C 0.000} C_DIS
LIN {X -10.461,Y -44.153,Z -226.669,A -90.000,B 90.000,C 0.000} C_DIS
LIN {X -10.221,Y -44.146,Z -227.004,A -90.000,B 90.000,C 0.000} C_DIS
LIN {X -9.986,Y -44.139,Z -227.363,A -90.000,B 90.000,C 0.000} C_DIS
LIN {X -9.672,Y -44.133,Z -227.879,A -90.000,B 90.000,C 0.000} C_DIS
LIN {X -9.243,Y -44.128,Z -228.589,A -90.000,B 90.000,C 0.000} C_DIS
LIN {X -8.940,Y -44.120,Z -229.090,A -90.000,B 90.000,C 0.000} C_DIS
LIN {X -8.341,Y -44.109,Z -230.112,A -90.000,B 90.000,C 0.000} C_DIS
LIN {X -8.151,Y -44.106,Z -230.463,A -90.000,B 90.000,C 0.000} C_DIS
LIN {X -8.082,Y -44.106,Z -230.600,A -90.000,B 90.000,C 0.000} C_DIS
LIN {X -7.936,Y -44.107,Z -230.901,A -90.000,B 90.000,C 0.000} C_DIS
LIN {X -7.634,Y -44.119,Z -231.573,A -90.000,B 90.000,C 0.000} C_DIS
LIN {X -7.588,Y -44.123,Z -231.675,A -90.000,B 90.000,C 0.000} C_DIS
LIN {X -6.420,Y -44.028,Z -231.267,A -90.000,B 90.000,C 0.000} C_DIS
LIN {X -6.098,Y -43.991,Z -230.999,A -90.000,B 90.000,C 0.000} C_DIS
LIN {X -5.414,Y -43.934,Z -230.427,A -90.000,B 90.000,C 0.000} C_DIS
LIN {X -5.007,Y -43.900,Z -230.087,A -90.000,B 90.000,C 0.000} C_DIS
LIN {X -4.512,Y -43.860,Z -229.688,A -90.000,B 90.000,C 0.000} C_DIS
LIN {X -4.346,Y -43.849,Z -229.554,A -90.000,B 90.000,C 0.000} C_DIS
LIN {X -2.258,Y -43.680,Z -227.122,A -90.000,B 90.000,C 0.000} C_DIS
LIN {X -1.919,Y -43.662,Z -226.725,A -90.000,B 90.000,C 0.000} C_DIS
LIN {X -0.490,Y -43.574,Z -224.638,A -90.000,B 90.000,C 0.000} C_DIS
LIN {X 0.691,Y -43.522,Z -222.906,A -90.000,B 90.000,C 0.000} C_DIS
LIN {X 1.002,Y -43.516,Z -222.451,A -90.000,B 90.000,C 0.000} C_DIS
LIN {X 1.298,Y -43.510,Z -222.023,A -90.000,B 90.000,C 0.000} C_DIS
LIN {X 2.819,Y -43.471,Z -219.523,A -90.000,B 90.000,C 0.000} C_DIS
LIN {X 3.643,Y -43.455,Z -218.166,A -90.000,B 90.000,C 0.000} C_DIS
LIN {X 3.797,Y -43.456,Z -217.911,A -90.000,B 90.000,C 0.000} C_DIS
LIN {X 5.331,Y -43.457,Z -215.179,A -90.000,B 90.000,C 0.000} C_DIS
LIN {X 6.269,Y -43.459,Z -213.557,A -90.000,B 90.000,C 0.000} C_DIS
LIN {X 7.092,Y -43.454,Z -211.982,A -90.000,B 90.000,C 0.000} C_DIS
LIN {X 7.490,Y -43.451,Z -211.191,A -90.000,B 90.000,C 0.000} C_DIS
LIN {X 8.409,Y -43.462,Z -209.357,A -90.000,B 90.000,C 0.000} C_DIS
LIN {X 8.564,Y -43.462,Z -209.031,A -90.000,B 90.000,C 0.000} C_DIS
LIN {X 8.864,Y -43.458,Z -208.318,A -90.000,B 90.000,C 0.000} C_DIS
LIN {X 9.818,Y -43.413,Z -206.047,A -90.000,B 90.000,C 0.000} C_DIS
LIN {X 9.994,Y -43.404,Z -205.611,A -90.000,B 90.000,C 0.000} C_DIS
LIN {X 10.053,Y -43.399,Z -205.443,A -90.000,B 90.000,C 0.000} C_DIS
LIN {X 10.652,Y -43.342,Z -203.739,A -90.000,B 90.000,C 0.000} C_DIS
LIN {X 10.905,Y -43.308,Z -202.911,A -90.000,B 90.000,C 0.000} C_DIS
LIN {X 10.905,Y -60.000,Z -202.911,A -90.000,B 90.000,C 0.000} C_DIS
LIN {X -16.911,Y -60.000,Z -219.601,A -90.000,B 90.000,C 0.000} C_DIS
LIN {X -16.911,Y -43.308,Z -219.601,A -90.000,B 90.000,C 0.000} C_DIS
LIN {X -16.844,Y -43.321,Z -219.622,A -90.000,B 90.000,C 0.000} C_DIS
LIN {X -16.725,Y -43.334,Z -219.664,A -90.000,B 90.000,C 0.000} C_DIS
LIN {X -16.394,Y -43.372,Z -219.790,A -90.000,B 90.000,C 0.000} C_DIS
LIN {X -15.952,Y -43.426,Z -219.977,A -90.000,B 90.000,C 0.000} C_DIS
LIN {X -15.617,Y -43.469,Z -220.131,A -90.000,B 90.000,C 0.000} C_DIS
LIN {X -15.337,Y -43.508,Z -220.271,A -90.000,B 90.000,C 0.000} C_DIS
LIN {X -15.009,Y -43.556,Z -220.448,A -90.000,B 90.000,C 0.000} C_DIS
LIN {X -14.726,Y -43.601,Z -220.609,A -90.000,B 90.000,C 0.000} C_DIS
LIN {X -14.504,Y -43.637,Z -220.743,A -90.000,B 90.000,C 0.000} C_DIS
LIN {X -14.179,Y -43.692,Z -220.950,A -90.000,B 90.000,C 0.000} C_DIS
LIN {X -13.840,Y -43.748,Z -221.179,A -90.000,B 90.000,C 0.000} C_DIS
LIN {X -13.179,Y -43.800,Z -221.636,A -90.000,B 90.000,C 0.000} C_DIS
LIN {X -12.543,Y -43.852,Z -222.081,A -90.000,B 90.000,C 0.000} C_DIS
LIN {X -11.669,Y -43.935,Z -222.725,A -90.000,B 90.000,C 0.000} C_DIS
LIN {X -11.568,Y -43.944,Z -222.801,A -90.000,B 90.000,C 0.000} C_DIS
LIN {X -11.402,Y -43.949,Z -222.926,A -90.000,B 90.000,C 0.000} C_DIS
LIN {X -11.189,Y -43.951,Z -223.089,A -90.000,B 90.000,C 0.000} C_DIS
LIN {X -10.855,Y -43.955,Z -223.361,A -90.000,B 90.000,C 0.000} C_DIS
LIN {X -10.431,Y -43.962,Z -223.734,A -90.000,B 90.000,C 0.000} C_DIS
LIN {X -10.397,Y -43.962,Z -223.765,A -90.000,B 90.000,C 0.000} C_DIS
LIN {X -10.237,Y -43.968,Z -223.915,A -90.000,B 90.000,C 0.000} C_DIS
LIN {X -10.015,Y -43.976,Z -224.133,A -90.000,B 90.000,C 0.000} C_DIS
LIN {X -9.810,Y -43.985,Z -224.347,A -90.000,B 90.000,C 0.000} C_DIS
LIN {X -9.476,Y -44.001,Z -224.716,A -90.000,B 90.000,C 0.000} C_DIS
LIN {X -9.359,Y -44.004,Z -224.852,A -90.000,B 90.000,C 0.000} C_DIS
LIN {X -9.087,Y -43.994,Z -225.184,A -90.000,B 90.000,C 0.000} C_DIS
LIN {X -8.836,Y -43.985,Z -225.514,A -90.000,B 90.000,C 0.000} C_DIS
LIN {X -8.555,Y -43.976,Z -225.910,A -90.000,B 90.000,C 0.000} C_DIS
LIN {X -8.287,Y -43.974,Z -226.320,A -90.000,B 90.000,C 0.000} C_DIS
LIN {X -7.854,Y -43.973,Z -227.034,A -90.000,B 90.000,C 0.000} C_DIS
LIN {X -7.222,Y -43.949,Z -228.081,A -90.000,B 90.000,C 0.000} C_DIS
LIN {X -6.870,Y -43.937,Z -228.683,A -90.000,B 90.000,C 0.000} C_DIS
LIN {X -6.730,Y -43.936,Z -228.921,A -90.000,B 90.000,C 0.000} C_DIS
LIN {X -6.262,Y -43.896,Z -228.530,A -90.000,B 90.000,C 0.000} C_DIS
LIN {X -5.744,Y -43.852,Z -228.112,A -90.000,B 90.000,C 0.000} C_DIS
LIN {X -3.905,Y -43.676,Z -225.970,A -90.000,B 90.000,C 0.000} C_DIS
LIN {X -3.511,Y -43.650,Z -225.511,A -90.000,B 90.000,C 0.000} C_DIS
LIN {X -2.800,Y -43.600,Z -224.473,A -90.000,B 90.000,C 0.000} C_DIS
LIN {X -2.140,Y -43.563,Z -223.508,A -90.000,B 90.000,C 0.000} C_DIS
LIN {X -0.932,Y -43.494,Z -221.738,A -90.000,B 90.000,C 0.000} C_DIS
LIN {X -0.380,Y -43.473,Z -220.935,A -90.000,B 90.000,C 0.000} C_DIS
LIN {X 1.419,Y -43.404,Z -217.978,A -90.000,B 90.000,C 0.000} C_DIS
LIN {X 2.083,Y -43.391,Z -216.880,A -90.000,B 90.000,C 0.000} C_DIS
LIN {X 2.249,Y -43.388,Z -216.584,A -90.000,B 90.000,C 0.000} C_DIS
LIN {X 3.603,Y -43.337,Z -214.179,A -90.000,B 90.000,C 0.000} C_DIS
LIN {X 4.394,Y -43.308,Z -212.816,A -90.000,B 90.000,C 0.000} C_DIS
LIN {X 4.394,Y -60.000,Z -212.816,A -90.000,B 90.000,C 0.000} C_DIS
LIN {X -13.778,Y -60.000,Z -218.871,A -90.000,B 90.000,C 0.000} C_DIS
LIN {X -13.778,Y -43.308,Z -218.871,A -90.000,B 90.000,C 0.000} C_DIS
LIN {X -13.494,Y -43.355,Z -219.041,A -90.000,B 90.000,C 0.000} C_DIS
LIN {X -13.378,Y -43.374,Z -219.111,A -90.000,B 90.000,C 0.000} C_DIS
LIN {X -13.031,Y -43.433,Z -219.333,A -90.000,B 90.000,C 0.000} C_DIS
LIN {X -12.545,Y -43.518,Z -219.660,A -90.000,B 90.000,C 0.000} C_DIS
LIN {X -12.270,Y -43.564,Z -219.847,A -90.000,B 90.000,C 0.000} C_DIS
LIN {X -11.737,Y -43.608,Z -220.218,A -90.000,B 90.000,C 0.000} C_DIS
LIN {X -11.348,Y -43.643,Z -220.490,A -90.000,B 90.000,C 0.000} C_DIS
LIN {X -10.188,Y -43.753,Z -221.348,A -90.000,B 90.000,C 0.000} C_DIS
LIN {X -10.014,Y -43.769,Z -221.480,A -90.000,B 90.000,C 0.000} C_DIS
LIN {X -9.908,Y -43.773,Z -221.563,A -90.000,B 90.000,C 0.000} C_DIS
LIN {X -9.600,Y -43.777,Z -221.815,A -90.000,B 90.000,C 0.000} C_DIS
LIN {X -9.526,Y -43.779,Z -221.877,A -90.000,B 90.000,C 0.000} C_DIS
LIN {X -9.067,Y -43.793,Z -222.280,A -90.000,B 90.000,C 0.000} C_DIS
LIN {X -8.820,Y -43.802,Z -222.514,A -90.000,B 90.000,C 0.000} C_DIS
LIN {X -8.573,Y -43.811,Z -222.756,A -90.000,B 90.000,C 0.000} C_DIS
LIN {X -8.315,Y -43.823,Z -223.028,A -90.000,B 90.000,C 0.000} C_DIS
LIN {X -8.015,Y -43.837,Z -223.359,A -90.000,B 90.000,C 0.000} C_DIS
LIN {X -7.872,Y -43.841,Z -223.524,A -90.000,B 90.000,C 0.000} C_DIS
LIN {X -7.818,Y -43.839,Z -223.588,A -90.000,B 90.000,C 0.000} C_DIS
LIN {X -7.568,Y -43.832,Z -223.893,A -90.000,B 90.000,C 0.000} C_DIS
LIN {X -7.510,Y -43.831,Z -223.965,A -90.000,B 90.000,C 0.000} C_DIS
LIN {X -7.212,Y -43.827,Z -224.358,A -90.000,B 90.000,C 0.000} C_DIS
LIN {X -6.930,Y -43.824,Z -224.754,A -90.000,B 90.000,C 0.000} C_DIS
LIN {X -6.763,Y -43.823,Z -225.007,A -90.000,B 90.000,C 0.000} C_DIS
LIN {X -6.583,Y -43.822,Z -225.284,A -90.000,B 90.000,C 0.000} C_DIS
LIN {X -6.380,Y -43.822,Z -225.620,A -90.000,B 90.000,C 0.000} C_DIS
LIN {X -6.321,Y -43.820,Z -225.716,A -90.000,B 90.000,C 0.000} C_DIS
LIN {X -5.491,Y -43.731,Z -224.748,A -90.000,B 90.000,C 0.000} C_DIS
LIN {X -5.098,Y -43.703,Z -224.290,A -90.000,B 90.000,C 0.000} C_DIS
LIN {X -3.385,Y -43.566,Z -221.784,A -90.000,B 90.000,C 0.000} C_DIS
LIN {X -2.528,Y -43.498,Z -220.529,A -90.000,B 90.000,C 0.000} C_DIS
LIN {X -2.060,Y -43.469,Z -219.848,A -90.000,B 90.000,C 0.000} C_DIS
LIN {X -0.985,Y -43.396,Z -218.080,A -90.000,B 90.000,C 0.000} C_DIS
LIN {X 0.041,Y -43.343,Z -216.394,A -90.000,B 90.000,C 0.000} C_DIS
LIN {X 0.371,Y -43.325,Z -215.846,A -90.000,B 90.000,C 0.000} C_DIS
LIN {X 0.660,Y -43.308,Z -215.333,A -90.000,B 90.000,C 0.000} C_DIS
LIN {X 0.660,Y -60.000,Z -215.333,A -90.000,B 90.000,C 0.000} C_DIS
LIN {X -11.243,Y -60.000,Z -218.144,A -90.000,B 90.000,C 0.000} C_DIS
LIN {X -11.243,Y -43.308,Z -218.144,A -90.000,B 90.000,C 0.000} C_DIS
LIN {X -10.803,Y -43.391,Z -218.444,A -90.000,B 90.000,C 0.000} C_DIS
LIN {X -10.727,Y -43.401,Z -218.496,A -90.000,B 90.000,C 0.000} C_DIS
LIN {X -10.153,Y -43.454,Z -218.898,A -90.000,B 90.000,C 0.000} C_DIS
LIN {X -9.101,Y -43.556,Z -219.675,A -90.000,B 90.000,C 0.000} C_DIS
LIN {X -8.780,Y -43.594,Z -219.916,A -90.000,B 90.000,C 0.000} C_DIS
LIN {X -8.630,Y -43.612,Z -220.033,A -90.000,B 90.000,C 0.000} C_DIS
LIN {X -8.307,Y -43.631,Z -220.295,A -90.000,B 90.000,C 0.000} C_DIS
LIN {X -8.208,Y -43.635,Z -220.380,A -90.000,B 90.000,C 0.000} C_DIS
LIN {X -7.695,Y -43.650,Z -220.832,A -90.000,B 90.000,C 0.000} C_DIS
LIN {X -7.417,Y -43.660,Z -221.095,A -90.000,B 90.000,C 0.000} C_DIS
LIN {X -7.126,Y -43.671,Z -221.383,A -90.000,B 90.000,C 0.000} C_DIS
LIN {X -7.000,Y -43.676,Z -221.516,A -90.000,B 90.000,C 0.000} C_DIS
LIN {X -6.833,Y -43.688,Z -221.691,A -90.000,B 90.000,C 0.000} C_DIS
LIN {X -6.469,Y -43.713,Z -222.095,A -90.000,B 90.000,C 0.000} C_DIS
LIN {X -6.386,Y -43.713,Z -222.191,A -90.000,B 90.000,C 0.000} C_DIS
LIN {X -6.275,Y -43.711,Z -222.322,A -90.000,B 90.000,C 0.000} C_DIS
LIN {X -6.220,Y -43.710,Z -222.389,A -90.000,B 90.000,C 0.000} C_DIS
LIN {X -5.289,Y -43.623,Z -221.026,A -90.000,B 90.000,C 0.000} C_DIS
LIN {X -4.608,Y -43.545,Z -220.029,A -90.000,B 90.000,C 0.000} C_DIS
LIN {X -4.180,Y -43.496,Z -219.402,A -90.000,B 90.000,C 0.000} C_DIS
LIN {X -3.740,Y -43.451,Z -218.761,A -90.000,B 90.000,C 0.000} C_DIS
LIN {X -3.574,Y -43.433,Z -218.488,A -90.000,B 90.000,C 0.000} C_DIS
LIN {X -2.315,Y -43.308,Z -216.421,A -90.000,B 90.000,C 0.000} C_DIS
LIN {X -2.278,Y -43.309,Z -216.356,A -90.000,B 90.000,C 0.000} C_DIS
LIN {X -2.207,Y -43.302,Z -216.231,A -90.000,B 90.000,C 0.000} C_DIS
LIN {X -2.142,Y -43.294,Z -216.109,A -90.000,B 90.000,C 0.000} C_DIS
LIN {X -2.083,Y -43.287,Z -215.990,A -90.000,B 90.000,C 0.000} C_DIS
LIN {X -2.007,Y -43.276,Z -215.817,A -90.000,B 90.000,C 0.000} C_DIS
LIN {X -1.964,Y -43.268,Z -215.705,A -90.000,B 90.000,C 0.000} C_DIS
LIN {X -1.927,Y -43.261,Z -215.596,A -90.000,B 90.000,C 0.000} C_DIS
LIN {X -1.882,Y -43.250,Z -215.438,A -90.000,B 90.000,C 0.000} C_DIS
LIN {X -1.859,Y -43.243,Z -215.337,A -90.000,B 90.000,C 0.000} C_DIS
LIN {X -1.842,Y -43.236,Z -215.238,A -90.000,B 90.000,C 0.000} C_DIS
LIN {X -1.830,Y -43.229,Z -215.142,A -90.000,B 90.000,C 0.000} C_DIS
LIN {X -1.824,Y -43.223,Z -215.049,A -90.000,B 90.000,C 0.000} C_DIS
LIN {X -1.823,Y -43.216,Z -214.958,A -90.000,B 90.000,C 0.000} C_DIS
LIN {X -1.827,Y -43.210,Z -214.870,A -90.000,B 90.000,C 0.000} C_DIS
LIN {X -1.836,Y -43.204,Z -214.785,A -90.000,B 90.000,C 0.000} C_DIS
LIN {X -1.850,Y -43.199,Z -214.703,A -90.000,B 90.000,C 0.000} C_DIS
LIN {X -1.869,Y -43.193,Z -214.622,A -90.000,B 90.000,C 0.000} C_DIS
LIN {X -1.893,Y -43.187,Z -214.545,A -90.000,B 90.000,C 0.000} C_DIS
LIN {X -1.920,Y -43.182,Z -214.470,A -90.000,B 90.000,C 0.000} C_DIS
LIN {X -1.953,Y -43.176,Z -214.398,A -90.000,B 90.000,C 0.000} C_DIS
LIN {X -1.989,Y -43.171,Z -214.329,A -90.000,B 90.000,C 0.000} C_DIS
LIN {X -2.030,Y -43.165,Z -214.262,A -90.000,B 90.000,C 0.000} C_DIS
LIN {X -2.076,Y -43.159,Z -214.199,A -90.000,B 90.000,C 0.000} C_DIS
LIN {X -2.125,Y -43.152,Z -214.137,A -90.000,B 90.000,C 0.000} C_DIS
LIN {X -2.179,Y -43.144,Z -214.078,A -90.000,B 90.000,C 0.000} C_DIS
LIN {X -2.267,Y -43.131,Z -213.994,A -90.000,B 90.000,C 0.000} C_DIS
LIN {X -2.330,Y -43.122,Z -213.942,A -90.000,B 90.000,C 0.000} C_DIS
LIN {X -2.398,Y -43.116,Z -213.893,A -90.000,B 90.000,C 0.000} C_DIS
LIN {X -2.542,Y -43.105,Z -213.799,A -90.000,B 90.000,C 0.000} C_DIS
LIN {X -2.699,Y -43.095,Z -213.715,A -90.000,B 90.000,C 0.000} C_DIS
LIN {X -2.868,Y -43.085,Z -213.641,A -90.000,B 90.000,C 0.000} C_DIS
LIN {X -3.048,Y -43.076,Z -213.575,A -90.000,B 90.000,C 0.000} C_DIS
LIN {X -3.239,Y -43.067,Z -213.519,A -90.000,B 90.000,C 0.000} C_DIS
LIN {X -3.439,Y -43.059,Z -213.472,A -90.000,B 90.000,C 0.000} C_DIS
LIN {X -3.648,Y -43.051,Z -213.433,A -90.000,B 90.000,C 0.000} C_DIS
LIN {X -3.865,Y -43.044,Z -213.403,A -90.000,B 90.000,C 0.000} C_DIS
LIN {X -3.976,Y -43.040,Z -213.391,A -90.000,B 90.000,C 0.000} C_DIS
LIN {X -4.203,Y -43.033,Z -213.373,A -90.000,B 90.000,C 0.000} C_DIS
LIN {X -4.436,Y -43.027,Z -213.364,A -90.000,B 90.000,C 0.000} C_DIS
LIN {X -4.673,Y -43.022,Z -213.362,A -90.000,B 90.000,C 0.000} C_DIS
LIN {X -4.914,Y -43.017,Z -213.368,A -90.000,B 90.000,C 0.000} C_DIS
LIN {X -5.282,Y -43.010,Z -213.392,A -90.000,B 90.000,C 0.000} C_DIS
LIN {X -5.529,Y -43.006,Z -213.417,A -90.000,B 90.000,C 0.000} C_DIS
LIN {X -5.777,Y -43.003,Z -213.449,A -90.000,B 90.000,C 0.000} C_DIS
LIN {X -6.025,Y -43.000,Z -213.488,A -90.000,B 90.000,C 0.000} C_DIS
LIN {X -6.395,Y -42.998,Z -213.559,A -90.000,B 90.000,C 0.000} C_DIS
LIN {X -6.760,Y -42.996,Z -213.646,A -90.000,B 90.000,C 0.000} C_DIS
LIN {X -6.999,Y -42.996,Z -213.711,A -90.000,B 90.000,C 0.000} C_DIS
LIN {X -7.234,Y -42.997,Z -213.783,A -90.000,B 90.000,C 0.000} C_DIS
LIN {X -7.463,Y -42.998,Z -213.861,A -90.000,B 90.000,C 0.000} C_DIS
LIN {X -7.796,Y -43.001,Z -213.989,A -90.000,B 90.000,C 0.000} C_DIS
LIN {X -8.009,Y -43.004,Z -214.081,A -90.000,B 90.000,C 0.000} C_DIS
LIN {X -8.213,Y -43.008,Z -214.179,A -90.000,B 90.000,C 0.000} C_DIS
LIN {X -8.408,Y -43.012,Z -214.282,A -90.000,B 90.000,C 0.000} C_DIS
LIN {X -8.594,Y -43.017,Z -214.390,A -90.000,B 90.000,C 0.000} C_DIS
LIN {X -8.768,Y -43.023,Z -214.503,A -90.000,B 90.000,C 0.000} C_DIS
LIN {X -8.930,Y -43.029,Z -214.621,A -90.000,B 90.000,C 0.000} C_DIS
LIN {X -9.080,Y -43.036,Z -214.743,A -90.000,B 90.000,C 0.000} C_DIS
LIN {X -9.217,Y -43.044,Z -214.870,A -90.000,B 90.000,C 0.000} C_DIS
LIN {X -9.339,Y -43.053,Z -215.001,A -90.000,B 90.000,C 0.000} C_DIS
LIN {X -9.446,Y -43.063,Z -215.137,A -90.000,B 90.000,C 0.000} C_DIS
LIN {X -9.493,Y -43.068,Z -215.206,A -90.000,B 90.000,C 0.000} C_DIS
LIN {X -9.536,Y -43.073,Z -215.276,A -90.000,B 90.000,C 0.000} C_DIS
LIN {X -9.575,Y -43.079,Z -215.347,A -90.000,B 90.000,C 0.000} C_DIS
LIN {X -9.610,Y -43.084,Z -215.419,A -90.000,B 90.000,C 0.000} C_DIS
LIN {X -9.640,Y -43.090,Z -215.492,A -90.000,B 90.000,C 0.000} C_DIS
LIN {X -9.666,Y -43.096,Z -215.566,A -90.000,B 90.000,C 0.000} C_DIS
LIN {X -9.687,Y -43.103,Z -215.641,A -90.000,B 90.000,C 0.000} C_DIS
LIN {X -9.703,Y -43.109,Z -215.716,A -90.000,B 90.000,C 0.000} C_DIS
LIN {X -9.718,Y -43.119,Z -215.831,A -90.000,B 90.000,C 0.000} C_DIS
LIN {X -9.721,Y -43.126,Z -215.909,A -90.000,B 90.000,C 0.000} C_DIS
LIN {X -9.720,Y -43.134,Z -215.987,A -90.000,B 90.000,C 0.000} C_DIS
LIN {X -9.708,Y -43.145,Z -216.106,A -90.000,B 90.000,C 0.000} C_DIS
LIN {X -9.693,Y -43.153,Z -216.186,A -90.000,B 90.000,C 0.000} C_DIS
LIN {X -9.672,Y -43.161,Z -216.267,A -90.000,B 90.000,C 0.000} C_DIS
LIN {X -9.631,Y -43.173,Z -216.390,A -90.000,B 90.000,C 0.000} C_DIS
LIN {X -9.596,Y -43.182,Z -216.472,A -90.000,B 90.000,C 0.000} C_DIS
LIN {X -9.555,Y -43.191,Z -216.555,A -90.000,B 90.000,C 0.000} C_DIS
LIN {X -9.483,Y -43.204,Z -216.681,A -90.000,B 90.000,C 0.000} C_DIS
LIN {X -9.427,Y -43.214,Z -216.766,A -90.000,B 90.000,C 0.000} C_DIS
LIN {X -9.364,Y -43.223,Z -216.851,A -90.000,B 90.000,C 0.000} C_DIS
LIN {X -9.259,Y -43.238,Z -216.980,A -90.000,B 90.000,C 0.000} C_DIS
LIN {X -9.138,Y -43.253,Z -217.110,A -90.000,B 90.000,C 0.000} C_DIS
LIN {X -9.050,Y -43.264,Z -217.197,A -90.000,B 90.000,C 0.000} C_DIS
LIN {X -8.850,Y -43.286,Z -217.371,A -90.000,B 90.000,C 0.000} C_DIS
LIN {X -8.625,Y -43.308,Z -217.550,A -90.000,B 90.000,C 0.000} C_DIS
LIN {X -8.473,Y -43.323,Z -217.662,A -90.000,B 90.000,C 0.000} C_DIS
LIN {X -7.894,Y -43.390,Z -218.090,A -90.000,B 90.000,C 0.000} C_DIS
LIN {X -7.541,Y -43.431,Z -218.354,A -90.000,B 90.000,C 0.000} C_DIS
LIN {X -7.344,Y -43.455,Z -218.509,A -90.000,B 90.000,C 0.000} C_DIS
LIN {X -7.148,Y -43.479,Z -218.667,A -90.000,B 90.000,C 0.000} C_DIS
LIN {X -6.982,Y -43.490,Z -218.803,A -90.000,B 90.000,C 0.000} C_DIS
LIN {X -6.796,Y -43.501,Z -218.965,A -90.000,B 90.000,C 0.000} C_DIS
LIN {X -6.488,Y -43.510,Z -219.236,A -90.000,B 90.000,C 0.000} C_DIS
LIN {X -5.738,Y -43.418,Z -218.139,A -90.000,B 90.000,C 0.000} C_DIS
LIN {X -5.421,Y -43.386,Z -217.678,A -90.000,B 90.000,C 0.000} C_DIS
LIN {X -5.093,Y -43.347,Z -217.140,A -90.000,B 90.000,C 0.000} C_DIS
LIN {X -4.784,Y -43.308,Z -216.633,A -90.000,B 90.000,C 0.000} C_DIS
LIN {X -4.784,Y -60.000,Z -216.633,A -90.000,B 90.000,C 0.000} C_DIS
LIN {X -69.214,Y -60.000,Z -243.561,A -90.000,B 90.000,C 0.000} C_DIS
LIN {X -69.214,Y -44.212,Z -243.561,A -90.000,B 90.000,C 0.000} C_DIS
LIN {X -69.177,Y -44.110,Z -243.356,A -90.000,B 90.000,C 0.000} C_DIS
LIN {X -69.152,Y -44.056,Z -243.242,A -90.000,B 90.000,C 0.000} C_DIS
LIN {X -69.134,Y -44.024,Z -243.176,A -90.000,B 90.000,C 0.000} C_DIS
LIN {X -68.983,Y -43.827,Z -242.733,A -90.000,B 90.000,C 0.000} C_DIS
LIN {X -68.898,Y -43.740,Z -242.526,A -90.000,B 90.000,C 0.000} C_DIS
LIN {X -68.766,Y -43.642,Z -242.275,A -90.000,B 90.000,C 0.000} C_DIS
LIN {X -68.611,Y -43.552,Z -242.028,A -90.000,B 90.000,C 0.000} C_DIS
LIN {X -68.544,Y -43.525,Z -241.940,A -90.000,B 90.000,C 0.000} C_DIS
LIN {X -68.170,Y -43.384,Z -241.478,A -90.000,B 90.000,C 0.000} C_DIS
LIN {X -68.089,Y -43.356,Z -241.383,A -90.000,B 90.000,C 0.000} C_DIS
LIN {X -68.013,Y -43.335,Z -241.303,A -90.000,B 90.000,C 0.000} C_DIS
LIN {X -67.887,Y -43.308,Z -241.187,A -90.000,B 90.000,C 0.000} C_DIS
LIN {X -67.758,Y -43.285,Z -241.066,A -90.000,B 90.000,C 0.000} C_DIS
LIN {X -67.642,Y -43.263,Z -240.964,A -90.000,B 90.000,C 0.000} C_DIS
LIN {X -67.449,Y -43.231,Z -240.804,A -90.000,B 90.000,C 0.000} C_DIS
LIN {X -67.372,Y -43.221,Z -240.747,A -90.000,B 90.000,C 0.000} C_DIS
LIN {X -67.279,Y -43.217,Z -240.688,A -90.000,B 90.000,C 0.000} C_DIS
LIN {X -67.232,Y -43.218,Z -240.664,A -90.000,B 90.000,C 0.000} C_DIS
LIN {X -67.196,Y -43.222,Z -240.653,A -90.000,B 90.000,C 0.000} C_DIS
LIN {X -67.182,Y -43.226,Z -240.652,A -90.000,B 90.000,C 0.000} C_DIS
LIN {X -67.163,Y -43.235,Z -240.658,A -90.000,B 90.000,C 0.000} C_DIS
LIN {X -67.154,Y -43.248,Z -240.676,A -90.000,B 90.000,C 0.000} C_DIS
LIN {X -67.154,Y -43.263,Z -240.705,A -90.000,B 90.000,C 0.000} C_DIS
LIN {X -67.165,Y -43.282,Z -240.744,A -90.000,B 90.000,C 0.000} C_DIS
LIN {X -67.184,Y -43.302,Z -240.792,A -90.000,B 90.000,C 0.000} C_DIS
LIN {X -67.250,Y -43.352,Z -240.915,A -90.000,B 90.000,C 0.000} C_DIS
LIN {X -67.295,Y -43.380,Z -240.989,A -90.000,B 90.000,C 0.000} C_DIS
LIN {X -67.347,Y -43.410,Z -241.071,A -90.000,B 90.000,C 0.000} C_DIS
LIN {X -67.472,Y -43.473,Z -241.254,A -90.000,B 90.000,C 0.000} C_DIS
LIN {X -67.706,Y -43.577,Z -241.572,A -90.000,B 90.000,C 0.000} C_DIS
LIN {X -67.889,Y -43.650,Z -241.806,A -90.000,B 90.000,C 0.000} C_DIS
LIN {X -68.196,Y -43.762,Z -242.179,A -90.000,B 90.000,C 0.000} C_DIS
LIN {X -68.418,Y -43.837,Z -242.436,A -90.000,B 90.000,C 0.000} C_DIS
LIN {X -68.649,Y -43.910,Z -242.695,A -90.000,B 90.000,C 0.000} C_DIS
LIN {X -68.887,Y -43.979,Z -242.952,A -90.000,B 90.000,C 0.000} C_DIS
LIN {X -69.129,Y -44.044,Z -243.202,A -90.000,B 90.000,C 0.000} C_DIS
LIN {X -69.371,Y -44.102,Z -243.440,A -90.000,B 90.000,C 0.000} C_DIS
LIN {X -69.610,Y -44.153,Z -243.663,A -90.000,B 90.000,C 0.000} C_DIS
LIN {X -69.844,Y -44.194,Z -243.867,A -90.000,B 90.000,C 0.000} C_DIS
LIN {X -70.068,Y -44.226,Z -244.046,A -90.000,B 90.000,C 0.000} C_DIS
LIN {X -70.177,Y -44.236,Z -244.123,A -90.000,B 90.000,C 0.000} C_DIS
LIN {X -70.282,Y -44.244,Z -244.195,A -90.000,B 90.000,C 0.000} C_DIS
LIN {X -70.382,Y -44.249,Z -244.258,A -90.000,B 90.000,C 0.000} C_DIS
LIN {X -70.525,Y -44.250,Z -244.337,A -90.000,B 90.000,C 0.000} C_DIS
LIN {X -70.614,Y -44.245,Z -244.377,A -90.000,B 90.000,C 0.000} C_DIS
LIN {X -70.657,Y -44.241,Z -244.393,A -90.000,B 90.000,C 0.000} C_DIS
LIN {X -70.738,Y -44.231,Z -244.419,A -90.000,B 90.000,C 0.000} C_DIS
LIN {X -70.777,Y -44.224,Z -244.427,A -90.000,B 90.000,C 0.000} C_DIS
LIN {X -70.849,Y -44.207,Z -244.436,A -90.000,B 90.000,C 0.000} C_DIS
LIN {X -70.883,Y -44.197,Z -244.436,A -90.000,B 90.000,C 0.000} C_DIS
LIN {X -70.915,Y -44.185,Z -244.433,A -90.000,B 90.000,C 0.000} C_DIS
LIN {X -70.975,Y -44.160,Z -244.419,A -90.000,B 90.000,C 0.000} C_DIS
LIN {X -71.027,Y -44.129,Z -244.391,A -90.000,B 90.000,C 0.000} C_DIS
LIN {X -71.050,Y -44.111,Z -244.372,A -90.000,B 90.000,C 0.000} C_DIS
LIN {X -71.092,Y -44.072,Z -244.324,A -90.000,B 90.000,C 0.000} C_DIS
LIN {X -71.126,Y -44.028,Z -244.261,A -90.000,B 90.000,C 0.000} C_DIS
LIN {X -71.151,Y -43.979,Z -244.185,A -90.000,B 90.000,C 0.000} C_DIS
LIN {X -71.167,Y -43.924,Z -244.094,A -90.000,B 90.000,C 0.000} C_DIS
LIN {X -71.171,Y -43.894,Z -244.042,A -90.000,B 90.000,C 0.000} C_DIS
LIN {X -71.173,Y -43.830,Z -243.925,A -90.000,B 90.000,C 0.000} C_DIS
LIN {X -71.164,Y -43.760,Z -243.792,A -90.000,B 90.000,C 0.000} C_DIS
LIN {X -71.145,Y -43.684,Z -243.643,A -90.000,B 90.000,C 0.000} C_DIS
LIN {X -71.130,Y -43.640,Z -243.561,A -90.000,B 90.000,C 0.000} C_DIS
LIN {X -71.092,Y -43.533,Z -243.343,A -90.000,B 90.000,C 0.000} C_DIS
LIN {X -71.059,Y -43.452,Z -243.179,A -90.000,B 90.000,C 0.000} C_DIS
LIN {X -71.025,Y -43.386,Z -243.038,A -90.000,B 90.000,C 0.000} C_DIS
LIN {X -70.978,Y -43.308,Z -242.880,A -90.000,B 90.000,C 0.000} C_DIS
LIN {X -70.978,Y -60.000,Z -242.880,A -90.000,B 90.000,C 0.000} C_DIS
LIN {X 51.831,Y -60.000,Z -140.334,A -90.000,B 90.000,C 0.000} C_DIS
LIN {X 51.831,Y -43.308,Z -140.334,A -90.000,B 90.000,C 0.000} C_DIS
LIN {X 52.232,Y -43.327,Z -140.008,A -90.000,B 90.000,C 0.000} C_DIS
LIN {X 52.611,Y -43.349,Z -139.715,A -90.000,B 90.000,C 0.000} C_DIS
LIN {X 52.781,Y -43.361,Z -139.592,A -90.000,B 90.000,C 0.000} C_DIS
LIN {X 53.582,Y -43.422,Z -139.036,A -90.000,B 90.000,C 0.000} C_DIS
LIN {X 53.895,Y -43.435,Z -138.784,A -90.000,B 90.000,C 0.000} C_DIS
LIN {X 54.053,Y -43.437,Z -138.660,A -90.000,B 90.000,C 0.000} C_DIS
LIN {X 54.310,Y -43.443,Z -138.466,A -90.000,B 90.000,C 0.000} C_DIS
LIN {X 54.479,Y -43.449,Z -138.347,A -90.000,B 90.000,C 0.000} C_DIS
LIN {X 54.753,Y -43.462,Z -138.165,A -90.000,B 90.000,C 0.000} C_DIS
LIN {X 54.946,Y -43.475,Z -138.046,A -90.000,B 90.000,C 0.000} C_DIS
LIN {X 56.343,Y -43.584,Z -137.220,A -90.000,B 90.000,C 0.000} C_DIS
LIN {X 56.839,Y -43.626,Z -136.927,A -90.000,B 90.000,C 0.000} C_DIS
LIN {X 57.770,Y -43.677,Z -136.386,A -90.000,B 90.000,C 0.000} C_DIS
LIN {X 58.060,Y -43.696,Z -136.229,A -90.000,B 90.000,C 0.000} C_DIS
LIN {X 58.208,Y -43.707,Z -136.154,A -90.000,B 90.000,C 0.000} C_DIS
LIN {X 58.366,Y -43.719,Z -136.077,A -90.000,B 90.000,C 0.000} C_DIS
LIN {X 58.554,Y -43.738,Z -135.986,A -90.000,B 90.000,C 0.000} C_DIS
LIN {X 58.741,Y -43.758,Z -135.902,A -90.000,B 90.000,C 0.000} C_DIS
LIN {X 59.645,Y -43.860,Z -135.516,A -90.000,B 90.000,C 0.000} C_DIS
LIN {X 59.927,Y -43.885,Z -135.400,A -90.000,B 90.000,C 0.000} C_DIS
LIN {X 60.200,Y -43.912,Z -135.300,A -90.000,B 90.000,C 0.000} C_DIS
LIN {X 60.591,Y -43.953,Z -135.170,A -90.000,B 90.000,C 0.000} C_DIS
LIN {X 62.125,Y -44.152,Z -134.654,A -90.000,B 90.000,C 0.000} C_DIS
LIN {X 62.291,Y -44.174,Z -134.601,A -90.000,B 90.000,C 0.000} C_DIS
LIN {X 62.570,Y -44.213,Z -134.521,A -90.000,B 90.000,C 0.000} C_DIS
LIN {X 62.745,Y -44.231,Z -134.477,A -90.000,B 90.000,C 0.000} C_DIS
LIN {X 62.933,Y -44.252,Z -134.437,A -90.000,B 90.000,C 0.000} C_DIS
LIN {X 63.290,Y -44.293,Z -134.371,A -90.000,B 90.000,C 0.000} C_DIS
LIN {X 63.388,Y -44.304,Z -134.356,A -90.000,B 90.000,C 0.000} C_DIS
LIN {X 63.563,Y -44.327,Z -134.336,A -90.000,B 90.000,C 0.000} C_DIS
LIN {X 63.685,Y -44.341,Z -134.324,A -90.000,B 90.000,C 0.000} C_DIS
LIN {X 63.804,Y -44.355,Z -134.316,A -90.000,B 90.000,C 0.000} C_DIS
LIN {X 63.975,Y -44.375,Z -134.310,A -90.000,B 90.000,C 0.000} C_DIS
LIN {X 64.172,Y -44.399,Z -134.306,A -90.000,B 90.000,C 0.000} C_DIS
LIN {X 65.149,Y -44.522,Z -134.326,A -90.000,B 90.000,C 0.000} C_DIS
LIN {X 65.281,Y -44.532,Z -134.330,A -90.000,B 90.000,C 0.000} C_DIS
LIN {X 65.887,Y -44.567,Z -134.350,A -90.000,B 90.000,C 0.000} C_DIS
LIN {X 65.999,Y -44.574,Z -134.359,A -90.000,B 90.000,C 0.000} C_DIS
LIN {X 66.317,Y -44.595,Z -134.395,A -90.000,B 90.000,C 0.000} C_DIS
LIN {X 66.446,Y -44.604,Z -134.414,A -90.000,B 90.000,C 0.000} C_DIS
LIN {X 66.602,Y -44.615,Z -134.443,A -90.000,B 90.000,C 0.000} C_DIS
LIN {X 66.953,Y -44.632,Z -134.509,A -90.000,B 90.000,C 0.000} C_DIS
LIN {X 67.188,Y -44.644,Z -134.562,A -90.000,B 90.000,C 0.000} C_DIS
LIN {X 67.322,Y -44.652,Z -134.599,A -90.000,B 90.000,C 0.000} C_DIS
LIN {X 67.536,Y -44.664,Z -134.667,A -90.000,B 90.000,C 0.000} C_DIS
LIN {X 67.707,Y -44.671,Z -134.725,A -90.000,B 90.000,C 0.000} C_DIS
LIN {X 67.885,Y -44.674,Z -134.785,A -90.000,B 90.000,C 0.000} C_DIS
LIN {X 67.960,Y -44.674,Z -134.810,A -90.000,B 90.000,C 0.000} C_DIS
LIN {X 68.952,Y -44.647,Z -135.154,A -90.000,B 90.000,C 0.000} C_DIS
LIN {X 69.021,Y -44.645,Z -135.180,A -90.000,B 90.000,C 0.000} C_DIS
LIN {X 69.262,Y -44.634,Z -135.277,A -90.000,B 90.000,C 0.000} C_DIS
LIN {X 69.480,Y -44.625,Z -135.376,A -90.000,B 90.000,C 0.000} C_DIS
LIN {X 69.604,Y -44.620,Z -135.438,A -90.000,B 90.000,C 0.000} C_DIS
LIN {X 69.977,Y -44.606,Z -135.643,A -90.000,B 90.000,C 0.000} C_DIS
LIN {X 70.083,Y -44.603,Z -135.707,A -90.000,B 90.000,C 0.000} C_DIS
LIN {X 70.222,Y -44.598,Z -135.796,A -90.000,B 90.000,C 0.000} C_DIS
LIN {X 70.500,Y -44.591,Z -135.986,A -90.000,B 90.000,C 0.000} C_DIS
LIN {X 70.614,Y -44.588,Z -136.071,A -90.000,B 90.000,C 0.000} C_DIS
LIN {X 70.734,Y -44.585,Z -136.165,A -90.000,B 90.000,C 0.000} C_DIS
LIN {X 70.818,Y -44.578,Z -136.233,A -90.000,B 90.000,C 0.000} C_DIS
LIN {X 71.023,Y -44.553,Z -136.406,A -90.000,B 90.000,C 0.000} C_DIS
LIN {X 71.147,Y -44.538,Z -136.518,A -90.000,B 90.000,C 0.000} C_DIS
LIN {X 71.343,Y -44.515,Z -136.713,A -90.000,B 90.000,C 0.000} C_DIS
LIN {X 71.974,Y -44.442,Z -137.377,A -90.000,B 90.000,C 0.000} C_DIS
LIN {X 72.128,Y -44.424,Z -137.549,A -90.000,B 90.000,C 0.000} C_DIS
LIN {X 72.179,Y -44.419,Z -137.609,A -90.000,B 90.000,C 0.000} C_DIS
LIN {X 72.374,Y -44.398,Z -137.847,A -90.000,B 90.000,C 0.000} C_DIS
LIN {X 72.432,Y -44.392,Z -137.920,A -90.000,B 90.000,C 0.000} C_DIS
LIN {X 72.610,Y -44.373,Z -138.163,A -90.000,B 90.000,C 0.000} C_DIS
LIN {X 72.752,Y -44.360,Z -138.375,A -90.000,B 90.000,C 0.000} C_DIS
LIN {X 72.855,Y -44.351,Z -138.541,A -90.000,B 90.000,C 0.000} C_DIS
LIN {X 73.291,Y -44.315,Z -139.297,A -90.000,B 90.000,C 0.000} C_DIS
LIN {X 73.600,Y -44.286,Z -139.769,A -90.000,B 90.000,C 0.000} C_DIS
LIN {X 73.844,Y -44.257,Z -140.141,A -90.000,B 90.000,C 0.000} C_DIS
LIN {X 73.897,Y -44.251,Z -140.228,A -90.000,B 90.000,C 0.000} C_DIS
LIN {X 74.011,Y -44.239,Z -140.426,A -90.000,B 90.000,C 0.000} C_DIS
LIN {X 74.147,Y -44.211,Z -140.684,A -90.000,B 90.000,C 0.000} C_DIS
LIN {X 74.201,Y -44.201,Z -140.792,A -90.000,B 90.000,C 0.000} C_DIS
LIN {X 74.267,Y -44.188,Z -140.929,A -90.000,B 90.000,C 0.000} C_DIS
LIN {X 74.310,Y -44.179,Z -141.027,A -90.000,B 90.000,C 0.000} C_DIS
LIN {X 74.972,Y -44.055,Z -142.621,A -90.000,B 90.000,C 0.000} C_DIS
LIN {X 75.034,Y -44.044,Z -142.786,A -90.000,B 90.000,C 0.000} C_DIS
LIN {X 75.155,Y -44.024,Z -143.143,A -90.000,B 90.000,C 0.000} C_DIS
LIN {X 75.212,Y -44.014,Z -143.333,A -90.000,B 90.000,C 0.000} C_DIS
LIN {X 75.518,Y -43.950,Z -144.503,A -90.000,B 90.000,C 0.000} C_DIS
LIN {X 75.537,Y -43.947,Z -144.586,A -90.000,B 90.000,C 0.000} C_DIS
LIN {X 75.603,Y -43.934,Z -144.891,A -90.000,B 90.000,C 0.000} C_DIS
LIN {X 75.633,Y -43.928,Z -145.062,A -90.000,B 90.000,C 0.000} C_DIS
LIN {X 75.687,Y -43.920,Z -145.425,A -90.000,B 90.000,C 0.000} C_DIS
LIN {X 75.792,Y -43.906,Z -146.275,A -90.000,B 90.000,C 0.000} C_DIS
LIN {X 75.890,Y -43.897,Z -147.050,A -90.000,B 90.000,C 0.000} C_DIS
LIN {X 76.150,Y -43.834,Z -149.200,A -90.000,B 90.000,C 0.000} C_DIS
LIN {X 76.185,Y -43.823,Z -149.580,A -90.000,B 90.000,C 0.000} C_DIS
LIN {X 76.200,Y -43.818,Z -149.822,A -90.000,B 90.000,C 0.000} C_DIS
LIN {X 76.238,Y -43.805,Z -150.959,A -90.000,B 90.000,C 0.000} C_DIS
LIN {X 76.244,Y -43.799,Z -151.168,A -90.000,B 90.000,C 0.000} C_DIS
LIN {X 76.272,Y -43.756,Z -152.269,A -90.000,B 90.000,C 0.000} C_DIS
LIN {X 76.317,Y -43.697,Z -153.699,A -90.000,B 90.000,C 0.000} C_DIS
LIN {X 76.317,Y -43.690,Z -153.927,A -90.000,B 90.000,C 0.000} C_DIS
LIN {X 76.312,Y -43.685,Z -154.149,A -90.000,B 90.000,C 0.000} C_DIS
LIN {X 76.276,Y -43.677,Z -154.838,A -90.000,B 90.000,C 0.000} C_DIS
LIN {X 76.087,Y -43.584,Z -158.062,A -90.000,B 90.000,C 0.000} C_DIS
LIN {X 76.048,Y -43.576,Z -158.502,A -90.000,B 90.000,C 0.000} C_DIS
LIN {X 76.007,Y -43.574,Z -158.810,A -90.000,B 90.000,C 0.000} C_DIS
LIN {X 75.913,Y -43.566,Z -159.401,A -90.000,B 90.000,C 0.000} C_DIS
LIN {X 75.849,Y -43.559,Z -159.801,A -90.000,B 90.000,C 0.000} C_DIS
LIN {X 75.321,Y -43.542,Z -162.611,A -90.000,B 90.000,C 0.000} C_DIS
LIN {X 75.279,Y -43.536,Z -162.808,A -90.000,B 90.000,C 0.000} C_DIS
LIN {X 75.252,Y -43.534,Z -162.922,A -90.000,B 90.000,C 0.000} C_DIS
LIN {X 75.186,Y -43.531,Z -163.173,A -90.000,B 90.000,C 0.000} C_DIS
LIN {X 74.344,Y -43.529,Z -166.096,A -90.000,B 90.000,C 0.000} C_DIS
LIN {X 74.115,Y -43.516,Z -166.875,A -90.000,B 90.000,C 0.000} C_DIS
